// TIA Portal V19 export
FUNCTION_BLOCK "A0301_Spintore_Lat_FB"   // FB59, LAD
TITLE = == GESTIONE DELLA STAZIONE P5 ==
// stored: MemoryReserve 100, SetENOAutomatically false
   VAR_INPUT
      AreaInterface { ExternalAccessible := 'False'; ExternalVisible := 'False'; ExternalWritable := 'False'} : "AreaInterface";
      ZSI { ExternalAccessible := 'False'; ExternalVisible := 'False'; ExternalWritable := 'False'} : "udt_ZoneSafetyInterface";
      DSI { ExternalAccessible := 'False'; ExternalVisible := 'False'; ExternalWritable := 'False'} : "udt_DeviceSafetyInterface";
      DataIn : Struct
         OP_Rest_PB : Bool;
         OP_Work_PB : Bool;
         Orz_1_AnalSens : Int;
         Orz_2_AnalSens : Int;
      END_STRUCT;
      CIn { ExternalAccessible := 'False'; ExternalVisible := 'False'; ExternalWritable := 'False'} : Struct
         Manager_SpinLat_1 : "ValveMachine_Manager";
         Manager_SpinLat_2 : "ValveMachine_Manager";
         Manager_Sollevatori : "ValveMachine_Manager";
         SemiAut_Pb : Bool;
         P4 : Struct
            Fermi : "ValveMachine_COut";
         END_STRUCT;
         P5 : Struct
            SpintoreLong : Struct   // Spintore Longitudinale
               Ax_Sts : Struct
                  PosAttesa_Reached : Bool;
                  PosFineSpinta_Reached : Bool;
               END_STRUCT;
               Spintore : "ValveMachine_COut";
               Ax : "Positioning_EPOS_Machine_COut";
               Vrt : "ValveMachine_COut";
               Orz : "ValveMachine_COut";
            END_STRUCT;
         END_STRUCT;
         Trasporto : "SpeedMachine_COut";
      END_STRUCT;
      Config : Struct
         Vrt_1 : "ValveMachine_Config";
         Orz_1 : "ValveMachine_Config";
         Vrt_2 : "ValveMachine_Config";
         Orz_2 : "ValveMachine_Config";
         Sollevatori : Array[1..7] of "ValveMachine_Config";
         QuotaIngombro_SpinLat2 : Real := 2700.0;
         QuotaIngombro_SpinLat1 { ExternalWritable := 'False'} : Real := 770.0;
         DelayMissingCondition : Time;
      END_STRUCT;
   END_VAR
   VAR_OUTPUT
      MachineInterface : "MachineInterface";
      COut : Struct
         Spin_Lat1 : Struct
            Standstill : Bool;
            Rest_CheckNext : Bool;
            Work_CheckNext : Bool;
            Rest : Bool;
            Work : Bool;
         END_STRUCT;
         Spin_Lat2 : Struct
            Standstill : Bool;
            Rest_CheckNext : Bool;
            Work_CheckNext : Bool;
            Rest : Bool;
            Work : Bool;
         END_STRUCT;
         Vrt_1 : "ValveMachine_COut";
         Orz_1 : "ValveMachine_COut";
         Vrt_2 : "ValveMachine_COut";
         Orz_2 : "ValveMachine_COut";
         Sollevatori : "ValveMachine_COut";
      END_STRUCT;
   END_VAR
   VAR_IN_OUT
      Spin_Lat_1 : Struct
         Par : "Analogic_SensorManagement_Par";
         Data : Struct
            Sens : "Analogic_SensorManagement_Data";
            HMI : "HMI_Preset";
         END_STRUCT;
         Par_Mach : "A0301_Mach_Sens_Par";
      END_STRUCT;
      Spin_Lat_2 : Struct
         Par : "Analogic_SensorManagement_Par";
         Data : Struct
            Sens : "Analogic_SensorManagement_Data";
            HMI : "HMI_Preset";
         END_STRUCT;
         Par_Mach : "A0301_Mach_Sens_Par";
      END_STRUCT;
   END_VAR
   VAR
      Alarm : Struct
         Vrt_1 : "ValveAlr";
         Orz_1 { S7_SetPoint := 'True'} : "ValveAlr";
         Orz_1_AnalSens_Issue : Bool;
         Vrt_2 : "ValveAlr";
         Orz_2 { S7_SetPoint := 'True'} : "ValveAlr";
         Orz_2_AnalSens_Issue : Bool;
         Sollevatori : Array[1..7] of "ValveAlr";
         Finestre : Struct
            SpinLat2_SpinLong_Stop : Bool;   // Allarme Spintore longitudinale a ridosso dello Spintore laterale 2 che non si è abbassato
            SpinLat1_SpinLong_Stop : Bool;   // Allarme Spintore longitudinale a ridosso dello Spintore laterale 1 che non si è abbassato
         END_STRUCT;
      END_STRUCT;
      Warning : Struct
         Vrt_1 : "ValveMachine_Wng";
         Orz_1 { S7_SetPoint := 'True'} : "ValveMachine_Wng";
         Orz_1_AnalSens { ExternalAccessible := 'False'; ExternalVisible := 'False'; ExternalWritable := 'False'} : "Analogic_SensorManagement_Warning";
         Vrt_2 : "ValveMachine_Wng";
         Orz_2 { S7_SetPoint := 'True'} : "ValveMachine_Wng";
         Orz_2_AnalSens { ExternalAccessible := 'False'; ExternalVisible := 'False'; ExternalWritable := 'False'} : "Analogic_SensorManagement_Warning";
         Sollevatori : Array[1..7] of "ValveMachine_Wng";
         Finestre : Struct
            SpinLat2_SpinLong_Stop : Bool;   // Allarme Spintore longitudinale a ridosso dello Spintore laterale 2 che non si è abbassato
            SpinLat1_SpinLong_Stop : Bool;   // Allarme Spintore longitudinale a ridosso dello Spintore laterale 1 che non si è abbassato
         END_STRUCT;
         OP_REST_MissingCnd : Bool;   // Mancanza comando arresto
         OP_WORK_MissingCnd : Bool;   // Mancanza consenso lavoro
      END_STRUCT;
      HMI : Struct
         Selection : Array[1..6] of Bool;   // 0=Disable / 1=Enable Pin
         Sollevatori_Sts { S7_SetPoint := 'True'} : "UDT_HMI-Sts_ValvePosA0301";
         "SpinLat1&2_Sts" { S7_SetPoint := 'True'} : "UDT_HMI-Sts_ValvePosA0301";
         "SpinLat1&2_Vrt_Sts" { S7_SetPoint := 'True'} : "UDT_HMI-Sts_ValvePosA0301";
         "SpinLat1&2_Orz_Sts" { S7_SetPoint := 'True'} : "UDT_HMI-Sts_ValvePosA0301";
         Orz_AnalSens_PB_Preset { ExternalAccessible := 'False'; ExternalVisible := 'False'; ExternalWritable := 'False'} : Bool;   // Pulsante Preset value
         Orz_AnalSens_Preset_Value : LReal;
      END_STRUCT;
      Sts : Struct
         "SpinLat1&2_Alarm" : Bool;
         "SpinLat1&2_Vrt_AlarmPresence" : Bool;
         "SpinLat1&2_Orz_AlarmPresence" : Bool;
         Sollevatori_AlarmPresence : Bool;
         OP_CanMoveFreely : Bool;
         OP_Rest_Cnd : Bool;
         Op_Work_Cnd : Bool;
         Beam : Struct
            H_B : Real;
            Len_Meas : Real;
            P_U_PLen : Real;
            P_L_PLen : Real;
         END_STRUCT;
         "En/Dis_SpinLat_2" : Bool;   // 1=Enable / 0=Disable
      END_STRUCT;
      Ctrl : Struct
         OP_Rest_Man : Bool;
         OP_Work_Man : Bool;
         OP_Rest_Aut : Bool;
         OP_Work_Aut : Bool;
         OP_Rest : Bool;
         OP_Work : Bool;
      END_STRUCT;
      Vrt_1 : "ValveMachine_FB";
      Orz_1 { S7_SetPoint := 'True'} : "ValveMachine_FB";
      Orz_1_AnalSens { S7_SetPoint := 'True'} : "Analogic_SensorManagement";
      Vrt_2 : "ValveMachine_FB";
      Orz_2 { S7_SetPoint := 'True'} : "ValveMachine_FB";
      Orz_2_AnalSens { S7_SetPoint := 'True'} : "Analogic_SensorManagement";
      Sollevatori : Array[1..6] of "ValveMachine_FB";
      AUX : Struct
         OP_Rest_PB : Bool;
         OP_Work_PB : Bool;
      END_STRUCT;
      TON_OP_REST_MissingCnd { S7_SetPoint := 'True'} : TON_TIME;
      TON_OP_WORK_MissingCnd { S7_SetPoint := 'True'} : TON_TIME;
      Finestre : Struct
         Quota_SpinLat2_Rest : Real;   // Quota per comando riposo SpintoreLaterale 2
         Quota_SpinLat1_Rest : Real;   // Quota per comando riposo SpintoreLaterale 1
         RestCnd_Vrt_1 : Bool;   // Spintore longitudinale a ridosso dello Spintore laterale 1 - Comando riposo
         RestCnd_Vrt_2 : Bool;   // Spintore longitudinale a ridosso dello Spintore laterale 2 - Comando riposo
      END_STRUCT;
   END_VAR
   VAR_TEMP
      PE : Struct
         OP_Rest_PB : Bool;
         OP_Work_PB : Bool;
      END_STRUCT;
   END_VAR
   VAR CONSTANT
      Offset_SpinLat2_Rest : Real := 50.0;   // Offset calcolato da quota ingombro Spintore Laterale2 per abbassarlo
      Offset_SpinLat1_Rest : Real := 50.0;   // Offset calcolato da quota ingombro Spintore Laterale1 per abbassarlo
   END_VAR
   VAR_TEMP   // added for the SCL form of the ladder/FBD networks
      _w1 : Bool;
      _w2 : Bool;
      _w3 : Bool;
      _w4 : Bool;
      _w5 : Bool;
      _w6 : Bool;
      _w7 : Bool;
      _w8 : Bool;
   END_VAR
BEGIN

REGION Network 1 (SCL): Reset allarmi
   IF #AreaInterface.RstAlarms THEN
       #Alarm.Orz_1_AnalSens_Issue := FALSE;
       #Alarm.Orz_2_AnalSens_Issue := FALSE;
   END_IF;

   IF #AreaInterface.RstAlarms AND #Vrt_2.COut.Rest AND #Orz_2.COut.Rest THEN
       #Alarm.Finestre.SpinLat2_SpinLong_Stop := 0;
       #Warning.Finestre.SpinLat2_SpinLong_Stop := 0;
   END_IF;

   IF #AreaInterface.RstAlarms AND #Vrt_1.COut.Rest AND #Orz_1.COut.Rest THEN
       #Alarm.Finestre.SpinLat1_SpinLong_Stop := 0;
       #Warning.Finestre.SpinLat1_SpinLong_Stop := 0;
   END_IF;
END_REGION

REGION Network 2: <+>
END_REGION

REGION Network 3: CONTROLLO -
END_REGION

REGION Network 4 (SCL): CONTROLLO - Finestre di ingombro & Controlli di posizione

   // Finestra ingombro SPINTORE LATERALE 2
   #Finestre.Quota_SpinLat2_Rest := #Config.QuotaIngombro_SpinLat2 - #Offset_SpinLat2_Rest;

   // Se ho lo Spintore longitudinale in movimento ed entro dentro la finestra abbasso lo Spintore laterale 2 prima di arrivarci addosso
   // //
   IF #Sts.Beam.Len_Meas <= 2700.0 THEN
       #Sts."En/Dis_SpinLat_2" := FALSE;

   ELSE
       #Sts."En/Dis_SpinLat_2" := TRUE;
       #Warning.Finestre.SpinLat2_SpinLong_Stop := FALSE;
   END_IF;

   //Se arrivo in quota ingombro spintore lat. 2 mando a riposo attivando il cmd finestra
   IF  #Finestre.Quota_SpinLat2_Rest <= #CIn.P5.SpintoreLong.Ax.ActualPosition THEN
       #Finestre.RestCnd_Vrt_2 := TRUE;
   ELSE
       #Finestre.RestCnd_Vrt_2 := FALSE;
   END_IF;

   // Se supero la quota di riposo Spintore Laterale 2 e non sono ancora a riposo con Spintore Laterale attivo warning
   IF #Finestre.Quota_SpinLat2_Rest < #CIn.P5.SpintoreLong.Ax.ActualPosition AND NOT #Vrt_2.COut.Rest THEN
       #Warning.Finestre.SpinLat2_SpinLong_Stop := TRUE;
   END_IF;

   //Se vado a riposo con spin. lat 2 resetto warning 
   IF (#Vrt_2.COut.Rest AND #Orz_2.COut.Rest) THEN
       #Warning.Finestre.SpinLat2_SpinLong_Stop := FALSE;
   END_IF;

   // Finestra ingombro SPINTORE LATERALE 1
   #Finestre.Quota_SpinLat1_Rest := #Config.QuotaIngombro_SpinLat1 - #Offset_SpinLat1_Rest;

   // Se ho lo Spintore longitudinale in movimento ed entro dentro la finestra abbasso lo Spintore laterale 1 prima di arrivarci addosso

   //Se arrivo in quota ingombro spintore lat. 1 mando a riposo attivando il cmd finestra 
   IF #Finestre.Quota_SpinLat1_Rest <= #CIn.P5.SpintoreLong.Ax.ActualPosition  THEN
       #Finestre.RestCnd_Vrt_1 := TRUE;
   ELSE
       #Finestre.RestCnd_Vrt_1 := FALSE;
   END_IF;

   // Se supero la quota di riposo Spintore Laterale 1 e non sono ancora a riposo con Spintore Laterale attivo warning
   IF #Finestre.Quota_SpinLat1_Rest < #CIn.P5.SpintoreLong.Ax.ActualPosition AND NOT #Vrt_1.COut.Rest THEN
       #Warning.Finestre.SpinLat1_SpinLong_Stop := TRUE;
   END_IF;

   //Se vado a riposo con spin. lat 2 resetto warning 
   IF (#Vrt_1.COut.Rest AND #Orz_1.COut.Rest) THEN
       #Warning.Finestre.SpinLat2_SpinLong_Stop := FALSE;

   END_IF;
END_REGION

REGION Network 5: <+>
END_REGION

REGION Network 6: Operazione può muoversi liberamente perchè non sposta nessun BEAM
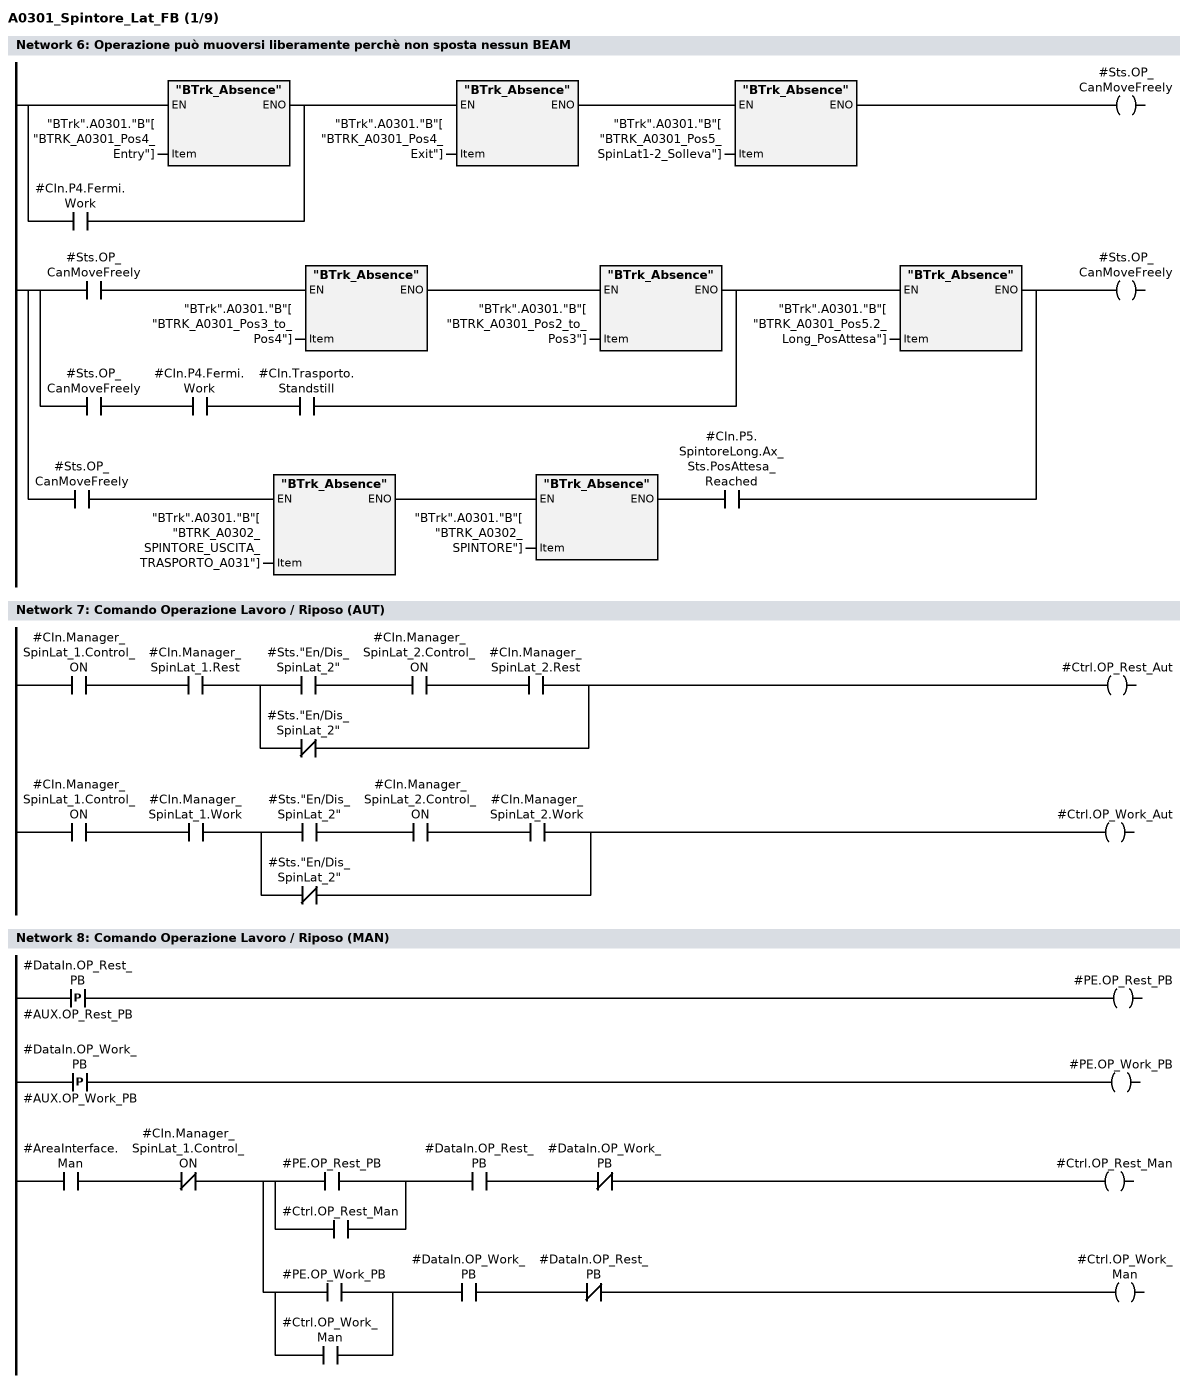
   RUNG wire#powerrail
      "BTrk_Absence"(Item := "BTrk".A0301."B"["BTRK_A0301_Pos4_Entry"])
      wire#w1
      "BTrk_Absence"(Item := "BTrk".A0301."B"["BTRK_A0301_Pos4_Exit"])
      "BTrk_Absence"(Item := "BTrk".A0301."B"["BTRK_A0301_Pos5_SpinLat1-2_Solleva"])
      Coil( #Sts.OP_CanMoveFreely )
   END_RUNG
   RUNG wire#powerrail
      Contact( #CIn.P4.Fermi.Work )
   END_RUNG wire#w1
   RUNG wire#powerrail
      Contact( #Sts.OP_CanMoveFreely )
      "BTrk_Absence"(Item := "BTrk".A0301."B"["BTRK_A0301_Pos3_to_Pos4"])
      "BTrk_Absence"(Item := "BTrk".A0301."B"["BTRK_A0301_Pos2_to_Pos3"])
      wire#w2
      "BTrk_Absence"(Item := "BTrk".A0301."B"["BTRK_A0301_Pos5.2_Long_PosAttesa"])
      wire#w3
      Coil( #Sts.OP_CanMoveFreely )
   END_RUNG
   RUNG wire#powerrail
      Contact( #Sts.OP_CanMoveFreely )
      Contact( #CIn.P4.Fermi.Work )
      Contact( #CIn.Trasporto.Standstill )
   END_RUNG wire#w2
   RUNG wire#powerrail
      Contact( #Sts.OP_CanMoveFreely )
      "BTrk_Absence"(Item := "BTrk".A0301."B"["BTRK_A0302_SPINTORE_USCITA_TRASPORTO_A031"])
      "BTrk_Absence"(Item := "BTrk".A0301."B"["BTRK_A0302_SPINTORE"])
      Contact( #CIn.P5.SpintoreLong.Ax_Sts.PosAttesa_Reached )
   END_RUNG wire#w3
   // the same network as SCL:
   "BTrk_Absence"(Item := "BTrk".A0301."B"["BTRK_A0301_Pos4_Entry"], ENO => #_w1);
   "BTrk_Absence"(EN := #_w1 OR #CIn.P4.Fermi.Work,
                  Item := "BTrk".A0301."B"["BTRK_A0301_Pos4_Exit"],
                  ENO => #_w2);
   "BTrk_Absence"(EN := #_w2, Item := "BTrk".A0301."B"["BTRK_A0301_Pos5_SpinLat1-2_Solleva"], ENO => #_w3);
   #Sts.OP_CanMoveFreely := #_w3;
   "BTrk_Absence"(EN := #Sts.OP_CanMoveFreely, Item := "BTrk".A0301."B"["BTRK_A0301_Pos3_to_Pos4"], ENO => #_w4);
   "BTrk_Absence"(EN := #_w4, Item := "BTrk".A0301."B"["BTRK_A0301_Pos2_to_Pos3"], ENO => #_w5);
   "BTrk_Absence"(EN := #_w5 OR (#Sts.OP_CanMoveFreely AND #CIn.P4.Fermi.Work AND #CIn.Trasporto.Standstill),
                  Item := "BTrk".A0301."B"["BTRK_A0301_Pos5.2_Long_PosAttesa"],
                  ENO => #_w6);
   "BTrk_Absence"(EN := #Sts.OP_CanMoveFreely,
                  Item := "BTrk".A0301."B"["BTRK_A0302_SPINTORE_USCITA_TRASPORTO_A031"],
                  ENO => #_w7);
   "BTrk_Absence"(EN := #_w7, Item := "BTrk".A0301."B"["BTRK_A0302_SPINTORE"], ENO => #_w8);
   #Sts.OP_CanMoveFreely := #_w6 OR (#_w8 AND #CIn.P5.SpintoreLong.Ax_Sts.PosAttesa_Reached);
END_REGION

REGION Network 7: Comando Operazione Lavoro / Riposo (AUT)
   RUNG wire#powerrail
      Contact( #CIn.Manager_SpinLat_1.Control_ON )
      Contact( #CIn.Manager_SpinLat_1.Rest )
      wire#w1
      Contact( #Sts."En/Dis_SpinLat_2" )
      Contact( #CIn.Manager_SpinLat_2.Control_ON )
      Contact( #CIn.Manager_SpinLat_2.Rest )
      wire#w2
      Coil( #Ctrl.OP_Rest_Aut )
   END_RUNG
   RUNG wire#w1
      I_Contact( #Sts."En/Dis_SpinLat_2" )
   END_RUNG wire#w2
   RUNG wire#powerrail
      Contact( #CIn.Manager_SpinLat_1.Control_ON )
      Contact( #CIn.Manager_SpinLat_1.Work )
      wire#w3
      Contact( #Sts."En/Dis_SpinLat_2" )
      Contact( #CIn.Manager_SpinLat_2.Control_ON )
      Contact( #CIn.Manager_SpinLat_2.Work )
      wire#w4
      Coil( #Ctrl.OP_Work_Aut )
   END_RUNG
   RUNG wire#w3
      I_Contact( #Sts."En/Dis_SpinLat_2" )
   END_RUNG wire#w4
   // the same network as SCL:
   #Ctrl.OP_Rest_Aut := #CIn.Manager_SpinLat_1.Control_ON AND #CIn.Manager_SpinLat_1.Rest AND ((#Sts."En/Dis_SpinLat_2" AND #CIn.Manager_SpinLat_2.Control_ON AND #CIn.Manager_SpinLat_2.Rest) OR NOT #Sts."En/Dis_SpinLat_2");
   #Ctrl.OP_Work_Aut := #CIn.Manager_SpinLat_1.Control_ON AND #CIn.Manager_SpinLat_1.Work AND ((#Sts."En/Dis_SpinLat_2" AND #CIn.Manager_SpinLat_2.Control_ON AND #CIn.Manager_SpinLat_2.Work) OR NOT #Sts."En/Dis_SpinLat_2");
END_REGION

REGION Network 8: Comando Operazione Lavoro / Riposo (MAN)
   RUNG wire#powerrail
      P_Contact(operand := #DataIn.OP_Rest_PB, bit := #AUX.OP_Rest_PB)
      Coil( #PE.OP_Rest_PB )
   END_RUNG
   RUNG wire#powerrail
      P_Contact(operand := #DataIn.OP_Work_PB, bit := #AUX.OP_Work_PB)
      Coil( #PE.OP_Work_PB )
   END_RUNG
   RUNG wire#powerrail
      Contact( #AreaInterface.Man )
      I_Contact( #CIn.Manager_SpinLat_1.Control_ON )
      wire#w1
      Contact( #PE.OP_Rest_PB )
      wire#w2
      Contact( #DataIn.OP_Rest_PB )
      I_Contact( #DataIn.OP_Work_PB )
      Coil( #Ctrl.OP_Rest_Man )
   END_RUNG
   RUNG wire#w1
      Contact( #Ctrl.OP_Rest_Man )
   END_RUNG wire#w2
   RUNG wire#w1
      Contact( #PE.OP_Work_PB )
      wire#w3
      Contact( #DataIn.OP_Work_PB )
      I_Contact( #DataIn.OP_Rest_PB )
      Coil( #Ctrl.OP_Work_Man )
   END_RUNG
   RUNG wire#w1
      Contact( #Ctrl.OP_Work_Man )
   END_RUNG wire#w3
   // the same network as SCL:
   #_w1 := #DataIn.OP_Rest_PB AND NOT #AUX.OP_Rest_PB;   // rising edge of #DataIn.OP_Rest_PB
   #AUX.OP_Rest_PB := #DataIn.OP_Rest_PB;
   #PE.OP_Rest_PB := #_w1;
   #_w2 := #DataIn.OP_Work_PB AND NOT #AUX.OP_Work_PB;   // rising edge of #DataIn.OP_Work_PB
   #AUX.OP_Work_PB := #DataIn.OP_Work_PB;
   #PE.OP_Work_PB := #_w2;
   #_w3 := #AreaInterface.Man AND NOT #CIn.Manager_SpinLat_1.Control_ON;
   #Ctrl.OP_Rest_Man := #_w3 AND (#PE.OP_Rest_PB OR #Ctrl.OP_Rest_Man) AND #DataIn.OP_Rest_PB AND NOT #DataIn.OP_Work_PB;
   #Ctrl.OP_Work_Man := #_w3 AND (#PE.OP_Work_PB OR #Ctrl.OP_Work_Man) AND #DataIn.OP_Work_PB AND NOT #DataIn.OP_Rest_PB;
END_REGION

REGION Network 9: Cumulativo Operazione Lavoro / Riposo (ALL)
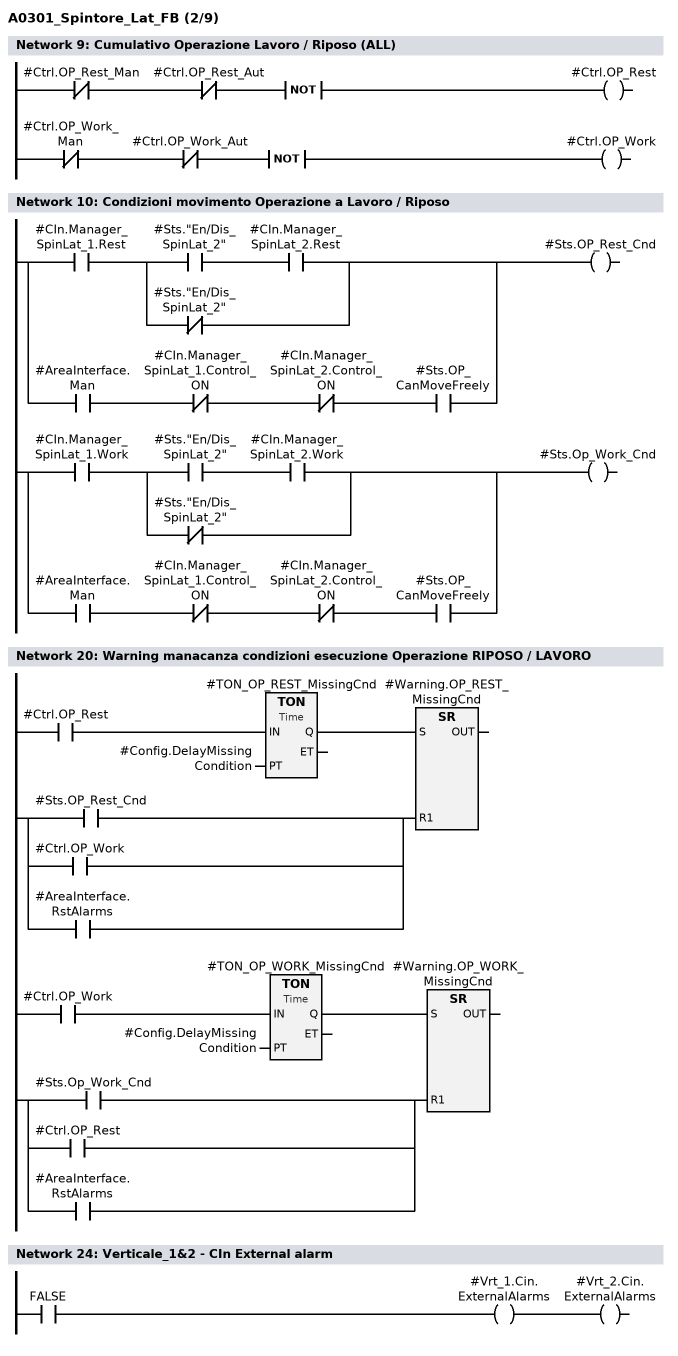
   RUNG wire#powerrail
      I_Contact( #Ctrl.OP_Rest_Man )
      I_Contact( #Ctrl.OP_Rest_Aut )
      Not()
      Coil( #Ctrl.OP_Rest )
   END_RUNG
   RUNG wire#powerrail
      I_Contact( #Ctrl.OP_Work_Man )
      I_Contact( #Ctrl.OP_Work_Aut )
      Not()
      Coil( #Ctrl.OP_Work )
   END_RUNG
   // the same network as SCL:
   #Ctrl.OP_Rest := NOT (NOT #Ctrl.OP_Rest_Man AND NOT #Ctrl.OP_Rest_Aut);
   #Ctrl.OP_Work := NOT (NOT #Ctrl.OP_Work_Man AND NOT #Ctrl.OP_Work_Aut);
END_REGION

REGION Network 10: Condizioni movimento Operazione a Lavoro / Riposo
   RUNG wire#powerrail
      Contact( #CIn.Manager_SpinLat_1.Rest )
      wire#w1
      Contact( #Sts."En/Dis_SpinLat_2" )
      Contact( #CIn.Manager_SpinLat_2.Rest )
      wire#w2
      Coil( #Sts.OP_Rest_Cnd )
   END_RUNG
   RUNG wire#w1
      I_Contact( #Sts."En/Dis_SpinLat_2" )
   END_RUNG wire#w2
   RUNG wire#powerrail
      Contact( #AreaInterface.Man )
      I_Contact( #CIn.Manager_SpinLat_1.Control_ON )
      I_Contact( #CIn.Manager_SpinLat_2.Control_ON )
      Contact( #Sts.OP_CanMoveFreely )
   END_RUNG wire#w2
   RUNG wire#powerrail
      Contact( #CIn.Manager_SpinLat_1.Work )
      wire#w3
      Contact( #Sts."En/Dis_SpinLat_2" )
      Contact( #CIn.Manager_SpinLat_2.Work )
      wire#w4
      Coil( #Sts.Op_Work_Cnd )
   END_RUNG
   RUNG wire#w3
      I_Contact( #Sts."En/Dis_SpinLat_2" )
   END_RUNG wire#w4
   RUNG wire#powerrail
      Contact( #AreaInterface.Man )
      I_Contact( #CIn.Manager_SpinLat_1.Control_ON )
      I_Contact( #CIn.Manager_SpinLat_2.Control_ON )
      Contact( #Sts.OP_CanMoveFreely )
   END_RUNG wire#w4
   // the same network as SCL:
   #Sts.OP_Rest_Cnd := (#CIn.Manager_SpinLat_1.Rest AND ((#Sts."En/Dis_SpinLat_2" AND #CIn.Manager_SpinLat_2.Rest) OR NOT #Sts."En/Dis_SpinLat_2")) OR (#AreaInterface.Man AND NOT #CIn.Manager_SpinLat_1.Control_ON AND NOT #CIn.Manager_SpinLat_2.Control_ON AND #Sts.OP_CanMoveFreely);
   #Sts.Op_Work_Cnd := (#CIn.Manager_SpinLat_1.Work AND ((#Sts."En/Dis_SpinLat_2" AND #CIn.Manager_SpinLat_2.Work) OR NOT #Sts."En/Dis_SpinLat_2")) OR (#AreaInterface.Man AND NOT #CIn.Manager_SpinLat_1.Control_ON AND NOT #CIn.Manager_SpinLat_2.Control_ON AND #Sts.OP_CanMoveFreely);
END_REGION

REGION Network 11: <+>
END_REGION

REGION Network 12 (SCL): Verticale + Orizzontale 1 - Cin Manager (Esecuzione sequenza comandi)
   #Vrt_1.Cin.Manager.Control_ON := #Orz_1.Cin.Manager.Control_ON := #CIn.Manager_SpinLat_1.Control_ON;

   #Vrt_1.Cin.Manager.Rest := FALSE;
   #Vrt_1.Cin.Manager.Work := FALSE;
   #Orz_1.Cin.Manager.Rest := FALSE;
   #Orz_1.Cin.Manager.Work := FALSE;


       IF (#Ctrl.OP_Rest AND #Sts.OP_Rest_Cnd) OR #Finestre.RestCnd_Vrt_1 THEN

           #Orz_1.Cin.Manager.Rest := #Vrt_1.Cin.Manager.Rest := TRUE;

       ELSIF (#Ctrl.OP_Work AND #Sts.Op_Work_Cnd) AND NOT #Finestre.RestCnd_Vrt_1 THEN

           #Orz_1.Cin.Manager.Work := #Vrt_1.Cin.Manager.Work := TRUE;

       END_IF;
END_REGION

REGION Network 13 (SCL): Verticale + Orizzontale1 - CIn Abilitazioni Stop Manager
   #Vrt_1.Cin.Manager.EnableStopDoorOpeningReq := #Orz_1.Cin.Manager.EnableStopDoorOpeningReq := #CIn.Manager_SpinLat_1.EnableStopDoorOpeningReq;

   #Vrt_1.Cin.Manager.EnableStopInPhase := #Orz_1.Cin.Manager.EnableStopInPhase := #CIn.Manager_SpinLat_1.EnableStopInPhase;

   #Vrt_1.Cin.Manager.EnableStopProgrammed := #Orz_1.Cin.Manager.EnableStopProgrammed := #CIn.Manager_SpinLat_1.EnableStopProgrammed;
END_REGION

REGION Network 14 (SCL): Verticale + Orizzontale 2 - Cin Manager (Esecuzione sequenza comandi)
   // Controllo della misura in lunghezza del Beam per sapere se abilitare il secondo spintore
   //
   #Vrt_2.Cin.Manager.Control_ON := #Orz_2.Cin.Manager.Control_ON := #CIn.Manager_SpinLat_2.Control_ON;
   //
   #Vrt_2.Cin.Manager.Rest := FALSE;
   #Vrt_2.Cin.Manager.Work := FALSE;
   #Orz_2.Cin.Manager.Rest := FALSE;
   #Orz_2.Cin.Manager.Work := FALSE;



   IF (#Ctrl.OP_Rest AND #Sts.OP_Rest_Cnd )OR #Finestre.RestCnd_Vrt_2 OR #Warning.Finestre.SpinLat2_SpinLong_Stop THEN

           #Orz_2.Cin.Manager.Rest := #Vrt_2.Cin.Manager.Rest := TRUE;

       ELSIF (#Ctrl.OP_Work AND #Sts.Op_Work_Cnd) AND #Sts."En/Dis_SpinLat_2" AND NOT #Finestre.RestCnd_Vrt_2  THEN

           #Orz_2.Cin.Manager.Work := #Vrt_2.Cin.Manager.Work := TRUE;

       END_IF;
END_REGION

REGION Network 15 (SCL): Verticale + Orizzontale 2 - CIn Abilitazioni Stop Manager
   #Vrt_2.Cin.Manager.EnableStopDoorOpeningReq := #Orz_2.Cin.Manager.EnableStopDoorOpeningReq := #CIn.Manager_SpinLat_2.EnableStopDoorOpeningReq;

   #Vrt_2.Cin.Manager.EnableStopInPhase := #Orz_2.Cin.Manager.EnableStopInPhase := #CIn.Manager_SpinLat_2.EnableStopInPhase;

   #Vrt_2.Cin.Manager.EnableStopProgrammed := #Orz_2.Cin.Manager.EnableStopProgrammed := #CIn.Manager_SpinLat_2.EnableStopProgrammed;
END_REGION

REGION Network 16: <+>
END_REGION

REGION Network 17 (SCL): S[1...7] Sollevatori - Cin Manager Comando arresto / lavoro
   //
   #Sollevatori[1].Cin.Manager.Rest := FALSE;
   #Sollevatori[2].Cin.Manager.Rest := FALSE;
   #Sollevatori[3].Cin.Manager.Rest := FALSE;
   #Sollevatori[4].Cin.Manager.Rest := FALSE;
   #Sollevatori[5].Cin.Manager.Rest := FALSE;
   #Sollevatori[6].Cin.Manager.Rest := FALSE;
   //************************************
   #Sollevatori[1].Cin.Manager.Work := FALSE;
   #Sollevatori[2].Cin.Manager.Work := FALSE;
   #Sollevatori[3].Cin.Manager.Work := FALSE;
   #Sollevatori[4].Cin.Manager.Work := FALSE;
   #Sollevatori[5].Cin.Manager.Work := FALSE;
   #Sollevatori[6].Cin.Manager.Work := FALSE;
   //
   // CIn Manager  Control ON se ho un richiesta di comando attiva
   IF #AreaInterface.Aut OR #CIn.SemiAut_Pb THEN
       #Sollevatori[1].Cin.Manager.Control_ON := TRUE;
       #Sollevatori[2].Cin.Manager.Control_ON := TRUE;
       #Sollevatori[3].Cin.Manager.Control_ON := TRUE;
       #Sollevatori[4].Cin.Manager.Control_ON := TRUE;
       #Sollevatori[5].Cin.Manager.Control_ON := TRUE;
       #Sollevatori[6].Cin.Manager.Control_ON := TRUE;
   ELSE
       #Sollevatori[1].Cin.Manager.Control_ON := FALSE;
       #Sollevatori[2].Cin.Manager.Control_ON := FALSE;
       #Sollevatori[3].Cin.Manager.Control_ON := FALSE;
       #Sollevatori[4].Cin.Manager.Control_ON := FALSE;
       #Sollevatori[5].Cin.Manager.Control_ON := FALSE;
       #Sollevatori[6].Cin.Manager.Control_ON := FALSE;
   END_IF;

   // CIn Manager Rest se ho un richiesta di comando arresto attiva
   IF #CIn.Manager_Sollevatori.Rest THEN

       #Sollevatori[1].Cin.Manager.Rest := TRUE;
       #Sollevatori[2].Cin.Manager.Rest := TRUE;
       #Sollevatori[3].Cin.Manager.Rest := TRUE;
       #Sollevatori[4].Cin.Manager.Rest := TRUE;
       #Sollevatori[5].Cin.Manager.Rest := TRUE;
       #Sollevatori[6].Cin.Manager.Rest := TRUE;

       // CIn Manager Work se ho un richiesta di comando lavoro attiva   
       ELSIF #CIn.Manager_Sollevatori.Work THEN

       #Sollevatori[1].Cin.Manager.Work := TRUE;
       #Sollevatori[2].Cin.Manager.Work := TRUE;
       #Sollevatori[3].Cin.Manager.Work := TRUE;
       #Sollevatori[4].Cin.Manager.Work := TRUE;
       #Sollevatori[5].Cin.Manager.Work := TRUE;
       #Sollevatori[6].Cin.Manager.Work := TRUE;

   END_IF;
END_REGION

REGION Network 18 (SCL): S[1...7] Sollevatori - CIn Abilitazioni Stop Manager
   //
   // CIn Manager Stop per richiesta apertura safety
   IF #CIn.Manager_SpinLat_1.EnableStopDoorOpeningReq THEN
       #Sollevatori[1].Cin.Manager.EnableStopDoorOpeningReq := TRUE;
       #Sollevatori[2].Cin.Manager.EnableStopDoorOpeningReq := TRUE;
       #Sollevatori[3].Cin.Manager.EnableStopDoorOpeningReq := TRUE;
       #Sollevatori[4].Cin.Manager.EnableStopDoorOpeningReq := TRUE;
       #Sollevatori[5].Cin.Manager.EnableStopDoorOpeningReq := TRUE;
       #Sollevatori[6].Cin.Manager.EnableStopDoorOpeningReq := TRUE;

   ELSE
       #Sollevatori[1].Cin.Manager.EnableStopDoorOpeningReq := FALSE;
       #Sollevatori[2].Cin.Manager.EnableStopDoorOpeningReq := FALSE;
       #Sollevatori[3].Cin.Manager.EnableStopDoorOpeningReq := FALSE;
       #Sollevatori[4].Cin.Manager.EnableStopDoorOpeningReq := FALSE;
       #Sollevatori[5].Cin.Manager.EnableStopDoorOpeningReq := FALSE;
       #Sollevatori[6].Cin.Manager.EnableStopDoorOpeningReq := FALSE;

   END_IF;
   // CIn Manager Stop in fase delle macchine precedenti
   IF #CIn.Manager_SpinLat_1.EnableStopInPhase THEN
       #Sollevatori[1].Cin.Manager.EnableStopInPhase := TRUE;
       #Sollevatori[2].Cin.Manager.EnableStopInPhase := TRUE;
       #Sollevatori[3].Cin.Manager.EnableStopInPhase := TRUE;
       #Sollevatori[4].Cin.Manager.EnableStopInPhase := TRUE;
       #Sollevatori[5].Cin.Manager.EnableStopInPhase := TRUE;
       #Sollevatori[6].Cin.Manager.EnableStopInPhase := TRUE;

   ELSE
       #Sollevatori[1].Cin.Manager.EnableStopInPhase := FALSE;
       #Sollevatori[2].Cin.Manager.EnableStopInPhase := FALSE;
       #Sollevatori[3].Cin.Manager.EnableStopInPhase := FALSE;
       #Sollevatori[4].Cin.Manager.EnableStopInPhase := FALSE;
       #Sollevatori[5].Cin.Manager.EnableStopInPhase := FALSE;
       #Sollevatori[6].Cin.Manager.EnableStopInPhase := FALSE;

   END_IF;

   // CIn Manager Stop programmato configurabile a piacere
   IF #CIn.Manager_SpinLat_1.EnableStopProgrammed THEN
       #Sollevatori[1].Cin.Manager.EnableStopProgrammed := TRUE;
       #Sollevatori[2].Cin.Manager.EnableStopProgrammed := TRUE;
       #Sollevatori[3].Cin.Manager.EnableStopProgrammed := TRUE;
       #Sollevatori[4].Cin.Manager.EnableStopProgrammed := TRUE;
       #Sollevatori[5].Cin.Manager.EnableStopProgrammed := TRUE;
       #Sollevatori[6].Cin.Manager.EnableStopProgrammed := TRUE;

   ELSE
       #Sollevatori[1].Cin.Manager.EnableStopProgrammed := FALSE;
       #Sollevatori[2].Cin.Manager.EnableStopProgrammed := FALSE;
       #Sollevatori[3].Cin.Manager.EnableStopProgrammed := FALSE;
       #Sollevatori[4].Cin.Manager.EnableStopProgrammed := FALSE;
       #Sollevatori[5].Cin.Manager.EnableStopProgrammed := FALSE;
       #Sollevatori[6].Cin.Manager.EnableStopProgrammed := FALSE;

   END_IF;
END_REGION

REGION Network 19: <+>
END_REGION

REGION Network 20: Warning manacanza condizioni esecuzione Operazione RIPOSO / LAVORO
   RUNG wire#powerrail
      Contact( #Ctrl.OP_Rest )
      { S7_Templates := "time_type := Time" } #TON_OP_REST_MissingCnd.TON(pt := #Config.DelayMissingCondition, et =>)
      S_SR(operand := #Warning.OP_REST_MissingCnd, r1 := wire#w1)
   END_RUNG
   RUNG wire#powerrail
      Contact( #Sts.OP_Rest_Cnd )
   END_RUNG wire#w1
   RUNG wire#powerrail
      Contact( #Ctrl.OP_Work )
   END_RUNG wire#w1
   RUNG wire#powerrail
      Contact( #AreaInterface.RstAlarms )
   END_RUNG wire#w1
   RUNG wire#powerrail
      Contact( #Ctrl.OP_Work )
      { S7_Templates := "time_type := Time" } #TON_OP_WORK_MissingCnd.TON(pt := #Config.DelayMissingCondition, et =>)
      S_SR(operand := #Warning.OP_WORK_MissingCnd, r1 := wire#w2)
   END_RUNG
   RUNG wire#powerrail
      Contact( #Sts.Op_Work_Cnd )
   END_RUNG wire#w2
   RUNG wire#powerrail
      Contact( #Ctrl.OP_Rest )
   END_RUNG wire#w2
   RUNG wire#powerrail
      Contact( #AreaInterface.RstAlarms )
   END_RUNG wire#w2
   // the same network as SCL:
   #TON_OP_REST_MissingCnd(IN := #Ctrl.OP_Rest, PT := #Config.DelayMissingCondition);   // TON
   IF #TON_OP_REST_MissingCnd.Q THEN
       #Warning.OP_REST_MissingCnd := TRUE;   // SR flip-flop
   END_IF;
   IF #Sts.OP_Rest_Cnd OR #Ctrl.OP_Work OR #AreaInterface.RstAlarms THEN
       #Warning.OP_REST_MissingCnd := FALSE;
   END_IF;
   #TON_OP_WORK_MissingCnd(IN := #Ctrl.OP_Work, PT := #Config.DelayMissingCondition);   // TON
   IF #TON_OP_WORK_MissingCnd.Q THEN
       #Warning.OP_WORK_MissingCnd := TRUE;   // SR flip-flop
   END_IF;
   IF #Sts.Op_Work_Cnd OR #Ctrl.OP_Rest OR #AreaInterface.RstAlarms THEN
       #Warning.OP_WORK_MissingCnd := FALSE;
   END_IF;
END_REGION

REGION Network 21: <+>
END_REGION

REGION Network 22: << GESTIONE VERTICALE >>
END_REGION

REGION Network 23 (SCL): Verticale1&2 - Data In
   // DataIn Scritti sulla CALL dell'FB
END_REGION

REGION Network 24: Verticale_1&2 - CIn External alarm
   RUNG wire#powerrail
      Contact( FALSE )
      Coil( #Vrt_1.Cin.ExternalAlarms )
      Coil( #Vrt_2.Cin.ExternalAlarms )
   END_RUNG
   // the same network as SCL:
   #Vrt_1.Cin.ExternalAlarms := FALSE;
   #Vrt_2.Cin.ExternalAlarms := FALSE;
END_REGION

REGION Network 25: Verticale_1 - Cin Ext Enable
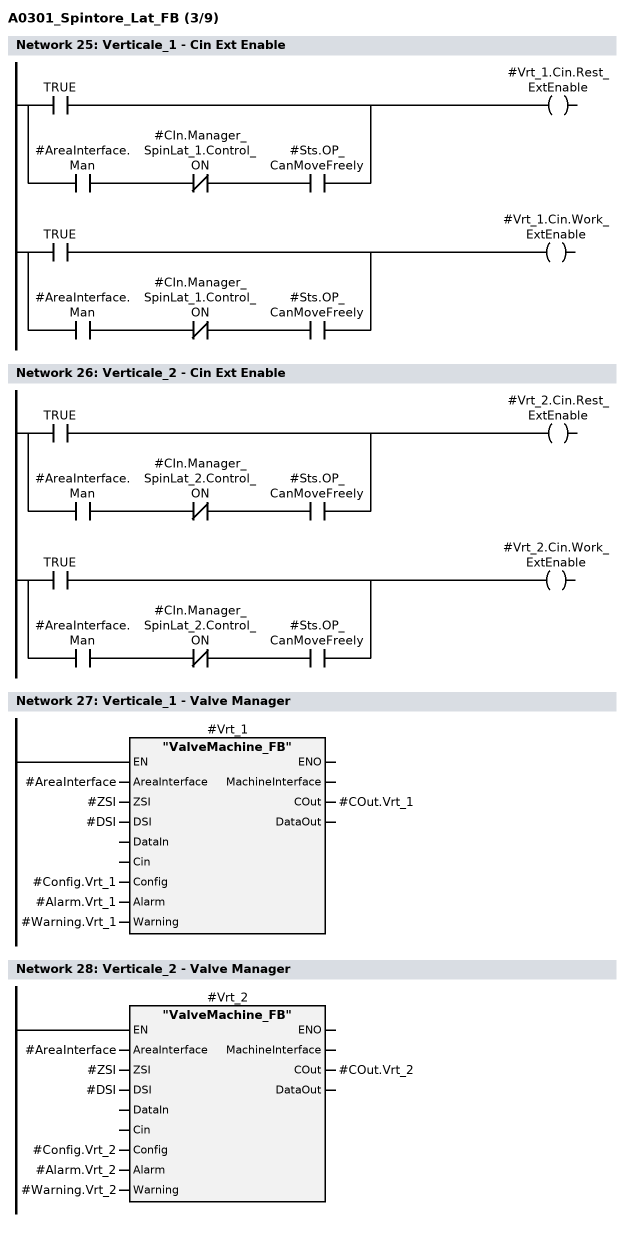
   RUNG wire#powerrail
      Contact( TRUE )
      wire#w1
      Coil( #Vrt_1.Cin.Rest_ExtEnable )
   END_RUNG
   RUNG wire#powerrail
      Contact( #AreaInterface.Man )
      I_Contact( #CIn.Manager_SpinLat_1.Control_ON )
      Contact( #Sts.OP_CanMoveFreely )
   END_RUNG wire#w1
   RUNG wire#powerrail
      Contact( TRUE )
      wire#w2
      Coil( #Vrt_1.Cin.Work_ExtEnable )
   END_RUNG
   RUNG wire#powerrail
      Contact( #AreaInterface.Man )
      I_Contact( #CIn.Manager_SpinLat_1.Control_ON )
      Contact( #Sts.OP_CanMoveFreely )
   END_RUNG wire#w2
   // the same network as SCL:
   #Vrt_1.Cin.Rest_ExtEnable := TRUE OR (#AreaInterface.Man AND NOT #CIn.Manager_SpinLat_1.Control_ON AND #Sts.OP_CanMoveFreely);
   #Vrt_1.Cin.Work_ExtEnable := TRUE OR (#AreaInterface.Man AND NOT #CIn.Manager_SpinLat_1.Control_ON AND #Sts.OP_CanMoveFreely);
END_REGION

REGION Network 26: Verticale_2 - Cin Ext Enable
   RUNG wire#powerrail
      Contact( TRUE )
      wire#w1
      Coil( #Vrt_2.Cin.Rest_ExtEnable )
   END_RUNG
   RUNG wire#powerrail
      Contact( #AreaInterface.Man )
      I_Contact( #CIn.Manager_SpinLat_2.Control_ON )
      Contact( #Sts.OP_CanMoveFreely )
   END_RUNG wire#w1
   RUNG wire#powerrail
      Contact( TRUE )
      wire#w2
      Coil( #Vrt_2.Cin.Work_ExtEnable )
   END_RUNG
   RUNG wire#powerrail
      Contact( #AreaInterface.Man )
      I_Contact( #CIn.Manager_SpinLat_2.Control_ON )
      Contact( #Sts.OP_CanMoveFreely )
   END_RUNG wire#w2
   // the same network as SCL:
   #Vrt_2.Cin.Rest_ExtEnable := TRUE OR (#AreaInterface.Man AND NOT #CIn.Manager_SpinLat_2.Control_ON AND #Sts.OP_CanMoveFreely);
   #Vrt_2.Cin.Work_ExtEnable := TRUE OR (#AreaInterface.Man AND NOT #CIn.Manager_SpinLat_2.Control_ON AND #Sts.OP_CanMoveFreely);
END_REGION

REGION Network 27: Verticale_1 - Valve Manager
   RUNG wire#powerrail
      #Vrt_1(AreaInterface := #AreaInterface, ZSI := #ZSI, DSI := #DSI, DataIn :=, Cin :=, Config := #Config.Vrt_1, Alarm := #Alarm.Vrt_1, Warning := #Warning.Vrt_1, MachineInterface =>, COut => #COut.Vrt_1, DataOut =>)
   END_RUNG
   // the same network as SCL:
   #Vrt_1(AreaInterface := #AreaInterface,   // "ValveMachine_FB"
          ZSI := #ZSI,
          DSI := #DSI,
          Config := #Config.Vrt_1,
          Alarm := #Alarm.Vrt_1,
          Warning := #Warning.Vrt_1,
          COut => #COut.Vrt_1);
END_REGION

REGION Network 28: Verticale_2 - Valve Manager
   RUNG wire#powerrail
      #Vrt_2(AreaInterface := #AreaInterface, ZSI := #ZSI, DSI := #DSI, DataIn :=, Cin :=, Config := #Config.Vrt_2, Alarm := #Alarm.Vrt_2, Warning := #Warning.Vrt_2, MachineInterface =>, COut => #COut.Vrt_2, DataOut =>)
   END_RUNG
   // the same network as SCL:
   #Vrt_2(AreaInterface := #AreaInterface,   // "ValveMachine_FB"
          ZSI := #ZSI,
          DSI := #DSI,
          Config := #Config.Vrt_2,
          Alarm := #Alarm.Vrt_2,
          Warning := #Warning.Vrt_2,
          COut => #COut.Vrt_2);
END_REGION

REGION Network 29: << GESTIONE ORIZZONTALE >>
END_REGION

REGION Network 30: <+>
END_REGION

REGION Network 31: << GESTIONE SPINTORE ORIZZ_1&2 - ANALOGIC SENSOR >>
END_REGION

REGION Network 33: Orizzontale_1 -Scalatura sensore
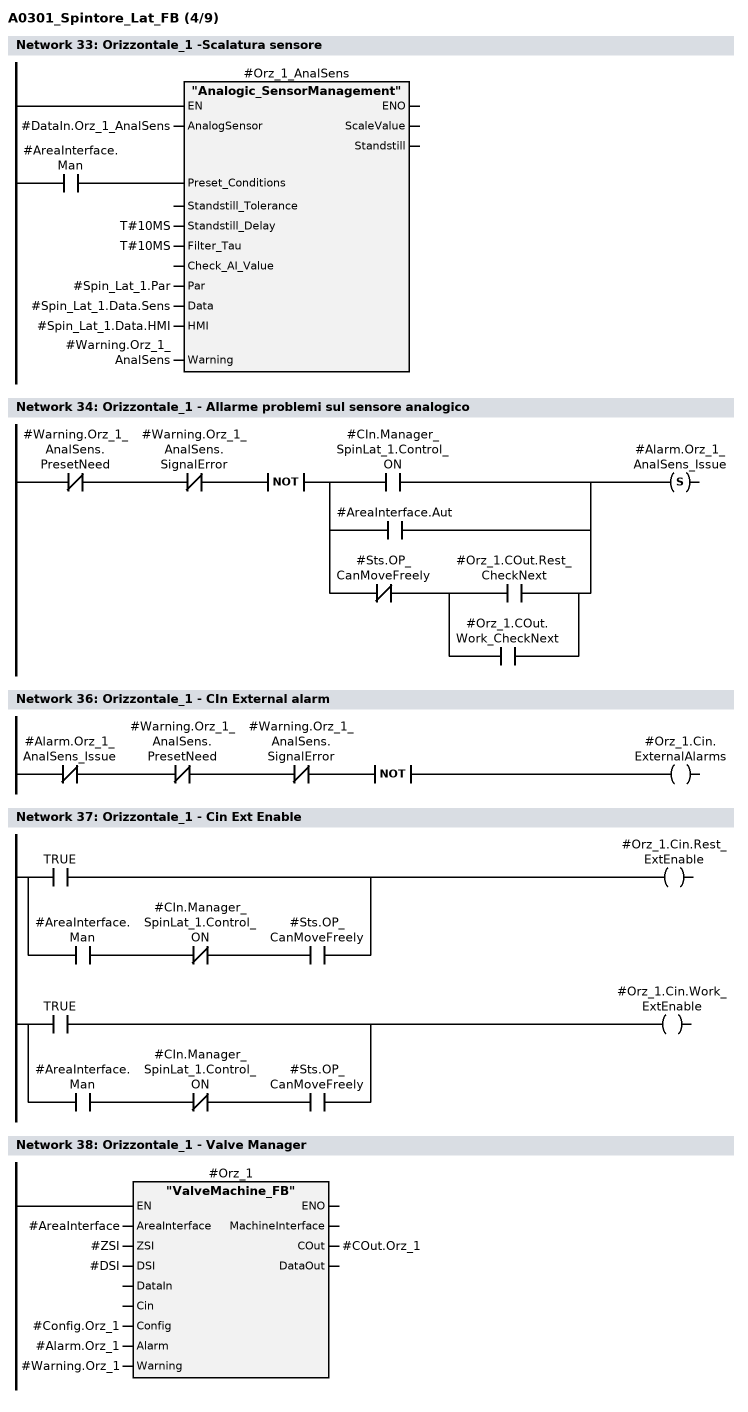
   RUNG wire#powerrail
      #Orz_1_AnalSens(Preset_Conditions := wire#w1, AnalogSensor := #DataIn.Orz_1_AnalSens, Standstill_Tolerance :=, Standstill_Delay := T#10MS, Filter_Tau := T#10MS, Check_AI_Value :=, Par := #Spin_Lat_1.Par, Data := #Spin_Lat_1.Data.Sens, HMI := #Spin_Lat_1.Data.HMI, Warning := #Warning.Orz_1_AnalSens, ScaleValue =>, Standstill =>)
   END_RUNG
   RUNG wire#powerrail
      Contact( #AreaInterface.Man )
   END_RUNG wire#w1
   // the same network as SCL:
   #Orz_1_AnalSens(AnalogSensor := #DataIn.Orz_1_AnalSens,   // "Analogic_SensorManagement"
                   Preset_Conditions := #AreaInterface.Man,
                   Standstill_Delay := T#10MS,
                   Filter_Tau := T#10MS,
                   Par := #Spin_Lat_1.Par,
                   Data := #Spin_Lat_1.Data.Sens,
                   HMI := #Spin_Lat_1.Data.HMI,
                   Warning := #Warning.Orz_1_AnalSens);
END_REGION

REGION Network 34: Orizzontale_1 - Allarme problemi sul sensore analogico
   RUNG wire#powerrail
      I_Contact( #Warning.Orz_1_AnalSens.PresetNeed )
      I_Contact( #Warning.Orz_1_AnalSens.SignalError )
      Not()
      wire#w1
      Contact( #CIn.Manager_SpinLat_1.Control_ON )
      wire#w2
      S_Coil( #Alarm.Orz_1_AnalSens_Issue )
   END_RUNG
   RUNG wire#w1
      Contact( #AreaInterface.Aut )
   END_RUNG wire#w2
   RUNG wire#w1
      I_Contact( #Sts.OP_CanMoveFreely )
      wire#w3
      Contact( #Orz_1.COut.Rest_CheckNext )
   END_RUNG wire#w2
   RUNG wire#w3
      Contact( #Orz_1.COut.Work_CheckNext )
   END_RUNG wire#w2
   // the same network as SCL:
   IF NOT (NOT #Warning.Orz_1_AnalSens.PresetNeed AND NOT #Warning.Orz_1_AnalSens.SignalError) AND (#CIn.Manager_SpinLat_1.Control_ON OR #AreaInterface.Aut OR (NOT #Sts.OP_CanMoveFreely AND (#Orz_1.COut.Rest_CheckNext OR #Orz_1.COut.Work_CheckNext))) THEN
       #Alarm.Orz_1_AnalSens_Issue := TRUE;
   END_IF;
END_REGION

REGION Network 35 (SCL): Orizzontale_1 - Datain / Config
   // DataIn Scritti sulla CALL dell'FB

   #Orz_1.Config := #Config.Orz_1;

   IF #Spin_Lat_1.Par.Enable AND #Sts.Beam.H_B > 0.0 THEN

       #Orz_1.DataIn.Work_Ls[1] := #Vrt_1.DataIn.Work_Ls[1] := ABS (#Orz_1_AnalSens.ScaleValue - #Sts.Beam.H_B) <= #Spin_Lat_1.Par_Mach.Tol_Work;
       #Orz_1.Config.V.WorkLimSwitchExist := TRUE;
       #Orz_1.Config.V.WorkTime := T#0.01s;

   ELSIF #Ctrl.OP_Rest THEN
       #Orz_1.DataIn.Work_Ls[1] := FALSE;
       #Vrt_1.DataIn.Work_Ls[1] := FALSE;

       // ********************************************************************************************************************************************
   ELSE
       // Overide della configurazione di default della valvola

       #Orz_1.Config.V.WorkLimSwitchExist := FALSE;
       #Orz_1.Config.V.WorkTime := #Spin_Lat_1.Par_Mach.WorkTime_SensDisable;
   END_IF;
END_REGION

REGION Network 36: Orizzontale_1 - CIn External alarm
   RUNG wire#powerrail
      I_Contact( #Alarm.Orz_1_AnalSens_Issue )
      I_Contact( #Warning.Orz_1_AnalSens.PresetNeed )
      I_Contact( #Warning.Orz_1_AnalSens.SignalError )
      Not()
      Coil( #Orz_1.Cin.ExternalAlarms )
   END_RUNG
   // the same network as SCL:
   #Orz_1.Cin.ExternalAlarms := NOT (NOT #Alarm.Orz_1_AnalSens_Issue AND NOT #Warning.Orz_1_AnalSens.PresetNeed AND NOT #Warning.Orz_1_AnalSens.SignalError);
END_REGION

REGION Network 37: Orizzontale_1 - Cin Ext Enable
   RUNG wire#powerrail
      Contact( TRUE )
      wire#w1
      Coil( #Orz_1.Cin.Rest_ExtEnable )
   END_RUNG
   RUNG wire#powerrail
      Contact( #AreaInterface.Man )
      I_Contact( #CIn.Manager_SpinLat_1.Control_ON )
      Contact( #Sts.OP_CanMoveFreely )
   END_RUNG wire#w1
   RUNG wire#powerrail
      Contact( TRUE )
      wire#w2
      Coil( #Orz_1.Cin.Work_ExtEnable )
   END_RUNG
   RUNG wire#powerrail
      Contact( #AreaInterface.Man )
      I_Contact( #CIn.Manager_SpinLat_1.Control_ON )
      Contact( #Sts.OP_CanMoveFreely )
   END_RUNG wire#w2
   // the same network as SCL:
   #Orz_1.Cin.Rest_ExtEnable := TRUE OR (#AreaInterface.Man AND NOT #CIn.Manager_SpinLat_1.Control_ON AND #Sts.OP_CanMoveFreely);
   #Orz_1.Cin.Work_ExtEnable := TRUE OR (#AreaInterface.Man AND NOT #CIn.Manager_SpinLat_1.Control_ON AND #Sts.OP_CanMoveFreely);
END_REGION

REGION Network 38: Orizzontale_1 - Valve Manager
   RUNG wire#powerrail
      #Orz_1(AreaInterface := #AreaInterface, ZSI := #ZSI, DSI := #DSI, DataIn :=, Cin :=, Config := #Config.Orz_1, Alarm := #Alarm.Orz_1, Warning := #Warning.Orz_1, MachineInterface =>, COut => #COut.Orz_1, DataOut =>)
   END_RUNG
   // the same network as SCL:
   #Orz_1(AreaInterface := #AreaInterface,   // "ValveMachine_FB"
          ZSI := #ZSI,
          DSI := #DSI,
          Config := #Config.Orz_1,
          Alarm := #Alarm.Orz_1,
          Warning := #Warning.Orz_1,
          COut => #COut.Orz_1);
END_REGION

REGION Network 39: <+>
END_REGION

REGION Network 40: Orizzontale_2 -Scalatura sensore
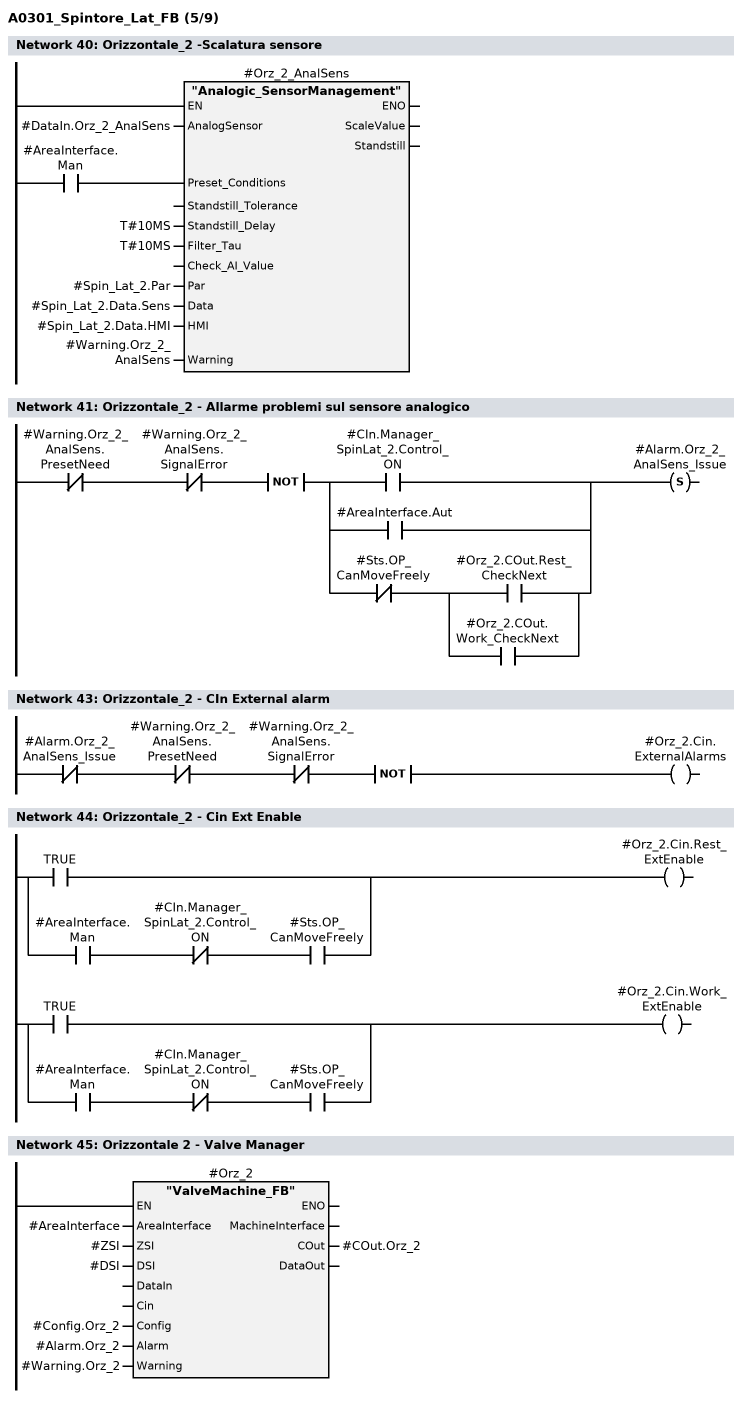
   RUNG wire#powerrail
      #Orz_2_AnalSens(Preset_Conditions := wire#w1, AnalogSensor := #DataIn.Orz_2_AnalSens, Standstill_Tolerance :=, Standstill_Delay := T#10MS, Filter_Tau := T#10MS, Check_AI_Value :=, Par := #Spin_Lat_2.Par, Data := #Spin_Lat_2.Data.Sens, HMI := #Spin_Lat_2.Data.HMI, Warning := #Warning.Orz_2_AnalSens, ScaleValue =>, Standstill =>)
   END_RUNG
   RUNG wire#powerrail
      Contact( #AreaInterface.Man )
   END_RUNG wire#w1
   // the same network as SCL:
   #Orz_2_AnalSens(AnalogSensor := #DataIn.Orz_2_AnalSens,   // "Analogic_SensorManagement"
                   Preset_Conditions := #AreaInterface.Man,
                   Standstill_Delay := T#10MS,
                   Filter_Tau := T#10MS,
                   Par := #Spin_Lat_2.Par,
                   Data := #Spin_Lat_2.Data.Sens,
                   HMI := #Spin_Lat_2.Data.HMI,
                   Warning := #Warning.Orz_2_AnalSens);
END_REGION

REGION Network 41: Orizzontale_2 - Allarme problemi sul sensore analogico
   RUNG wire#powerrail
      I_Contact( #Warning.Orz_2_AnalSens.PresetNeed )
      I_Contact( #Warning.Orz_2_AnalSens.SignalError )
      Not()
      wire#w1
      Contact( #CIn.Manager_SpinLat_2.Control_ON )
      wire#w2
      S_Coil( #Alarm.Orz_2_AnalSens_Issue )
   END_RUNG
   RUNG wire#w1
      Contact( #AreaInterface.Aut )
   END_RUNG wire#w2
   RUNG wire#w1
      I_Contact( #Sts.OP_CanMoveFreely )
      wire#w3
      Contact( #Orz_2.COut.Rest_CheckNext )
   END_RUNG wire#w2
   RUNG wire#w3
      Contact( #Orz_2.COut.Work_CheckNext )
   END_RUNG wire#w2
   // the same network as SCL:
   IF NOT (NOT #Warning.Orz_2_AnalSens.PresetNeed AND NOT #Warning.Orz_2_AnalSens.SignalError) AND (#CIn.Manager_SpinLat_2.Control_ON OR #AreaInterface.Aut OR (NOT #Sts.OP_CanMoveFreely AND (#Orz_2.COut.Rest_CheckNext OR #Orz_2.COut.Work_CheckNext))) THEN
       #Alarm.Orz_2_AnalSens_Issue := TRUE;
   END_IF;
END_REGION

REGION Network 42 (SCL): Orizzontale_2 - Datain / Config
   // DataIn Scritti sulla CALL dell'FB
   #Orz_2.Config := #Config.Orz_2;
   #Spin_Lat_2.Par.Enable := TRUE;

   // Se dal controllo di misura la lunghezza del Beam supera la Quota di abilitazione Spintore 2 abilito il controllo del sensore compensatore sul cilindro ORZ
   IF #Sts."En/Dis_SpinLat_2" THEN

   // *******************************************************************************************************************
   IF  #Spin_Lat_2.Par.Enable AND #Sts.Beam.H_B > 0.0 THEN
       #Spin_Lat_2.Par_Mach.Tol_Work := #Spin_Lat_1.Par_Mach.Tol_Work;

       #Orz_2.DataIn.Work_Ls[1] := #Vrt_2.DataIn.Work_Ls[1] := ABS (#Orz_2_AnalSens.ScaleValue - #Sts.Beam.H_B) <= #Spin_Lat_2.Par_Mach.Tol_Work;
       #Orz_2.Config.V.WorkLimSwitchExist := TRUE;
       #Orz_2.Config.V.WorkTime := T#0.01s;

   ELSIF #Ctrl.OP_Rest THEN
       #Orz_2.DataIn.Work_Ls[1] := FALSE;
       #Vrt_2.DataIn.Work_Ls[1] := FALSE;

       // ***************************************************************************************************************
   ELSE
       // Overide della configurazione di default della valvola

       #Orz_2.DataIn.Work_Ls[1] := FALSE;
       #Orz_2.Config.V.WorkLimSwitchExist := FALSE;
       #Orz_2.Config.V.WorkTime := #Spin_Lat_2.Par_Mach.WorkTime_SensDisable;
   END_IF;
   END_IF;
END_REGION

REGION Network 43: Orizzontale_2 - CIn External alarm
   RUNG wire#powerrail
      I_Contact( #Alarm.Orz_2_AnalSens_Issue )
      I_Contact( #Warning.Orz_2_AnalSens.PresetNeed )
      I_Contact( #Warning.Orz_2_AnalSens.SignalError )
      Not()
      Coil( #Orz_2.Cin.ExternalAlarms )
   END_RUNG
   // the same network as SCL:
   #Orz_2.Cin.ExternalAlarms := NOT (NOT #Alarm.Orz_2_AnalSens_Issue AND NOT #Warning.Orz_2_AnalSens.PresetNeed AND NOT #Warning.Orz_2_AnalSens.SignalError);
END_REGION

REGION Network 44: Orizzontale_2 - Cin Ext Enable
   RUNG wire#powerrail
      Contact( TRUE )
      wire#w1
      Coil( #Orz_2.Cin.Rest_ExtEnable )
   END_RUNG
   RUNG wire#powerrail
      Contact( #AreaInterface.Man )
      I_Contact( #CIn.Manager_SpinLat_2.Control_ON )
      Contact( #Sts.OP_CanMoveFreely )
   END_RUNG wire#w1
   RUNG wire#powerrail
      Contact( TRUE )
      wire#w2
      Coil( #Orz_2.Cin.Work_ExtEnable )
   END_RUNG
   RUNG wire#powerrail
      Contact( #AreaInterface.Man )
      I_Contact( #CIn.Manager_SpinLat_2.Control_ON )
      Contact( #Sts.OP_CanMoveFreely )
   END_RUNG wire#w2
   // the same network as SCL:
   #Orz_2.Cin.Rest_ExtEnable := TRUE OR (#AreaInterface.Man AND NOT #CIn.Manager_SpinLat_2.Control_ON AND #Sts.OP_CanMoveFreely);
   #Orz_2.Cin.Work_ExtEnable := TRUE OR (#AreaInterface.Man AND NOT #CIn.Manager_SpinLat_2.Control_ON AND #Sts.OP_CanMoveFreely);
END_REGION

REGION Network 45: Orizzontale 2 - Valve Manager
   RUNG wire#powerrail
      #Orz_2(AreaInterface := #AreaInterface, ZSI := #ZSI, DSI := #DSI, DataIn :=, Cin :=, Config := #Config.Orz_2, Alarm := #Alarm.Orz_2, Warning := #Warning.Orz_2, MachineInterface =>, COut => #COut.Orz_2, DataOut =>)
   END_RUNG
   // the same network as SCL:
   #Orz_2(AreaInterface := #AreaInterface,   // "ValveMachine_FB"
          ZSI := #ZSI,
          DSI := #DSI,
          Config := #Config.Orz_2,
          Alarm := #Alarm.Orz_2,
          Warning := #Warning.Orz_2,
          COut => #COut.Orz_2);
END_REGION

REGION Network 47: << GESTIONE SOLLEVATORI >>
END_REGION

REGION Network 48: S[1...6] Sollevatori - CIn External alarm
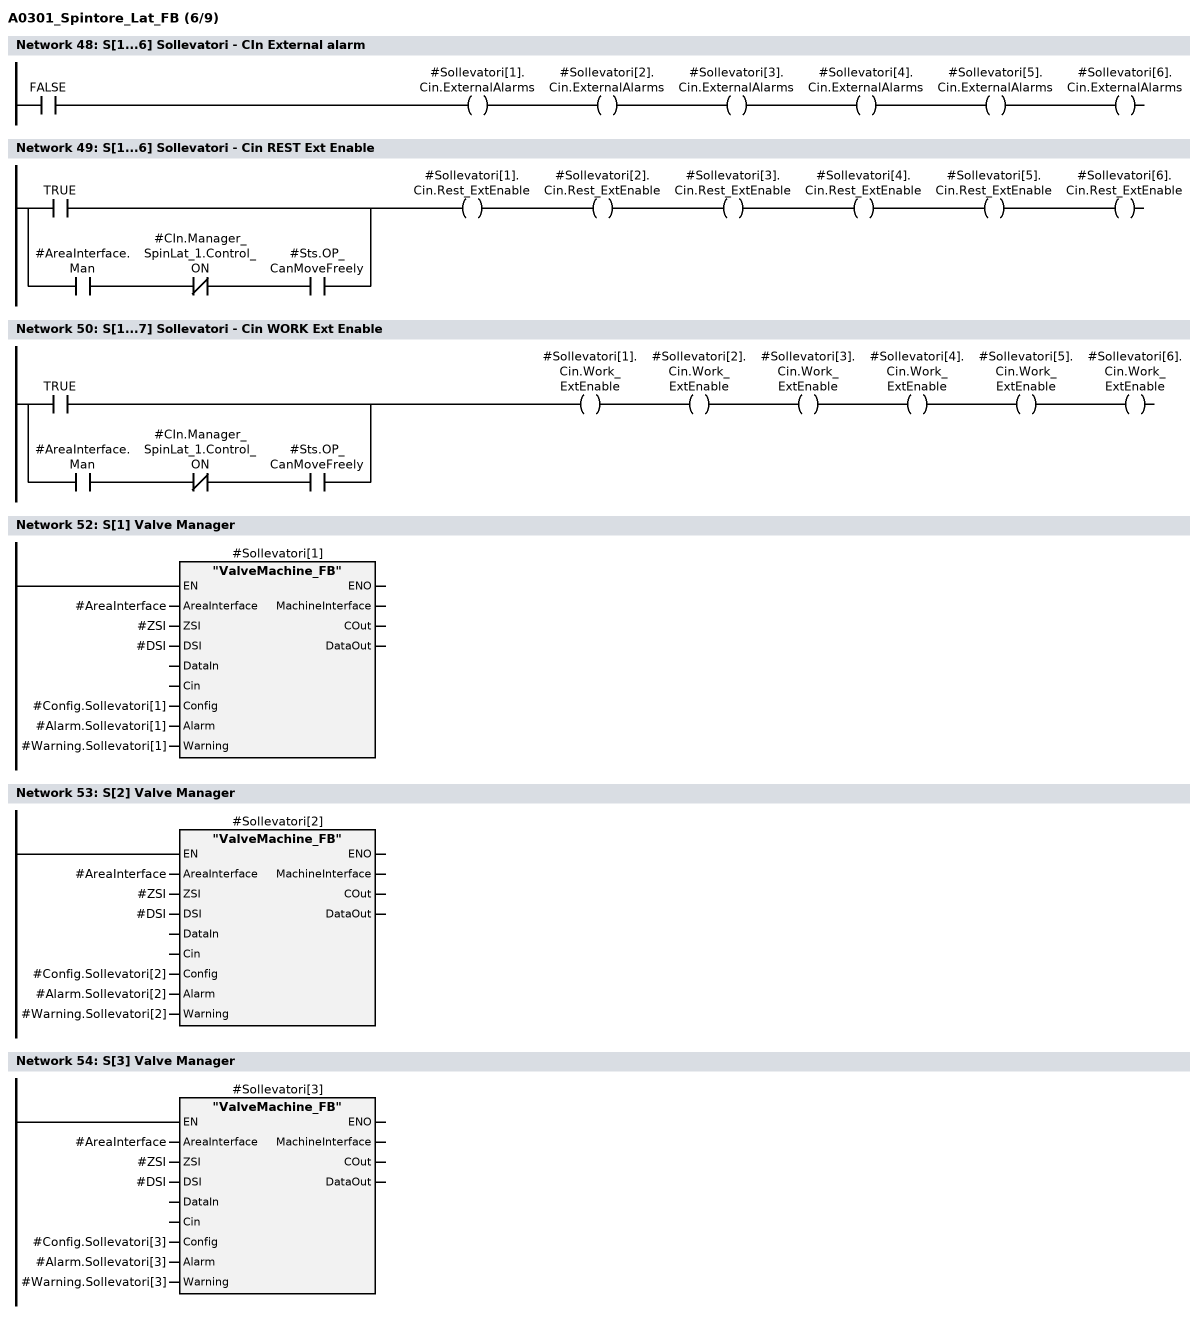
   RUNG wire#powerrail
      Contact( FALSE )
      Coil( #Sollevatori[1].Cin.ExternalAlarms )
      Coil( #Sollevatori[2].Cin.ExternalAlarms )
      Coil( #Sollevatori[3].Cin.ExternalAlarms )
      Coil( #Sollevatori[4].Cin.ExternalAlarms )
      Coil( #Sollevatori[5].Cin.ExternalAlarms )
      Coil( #Sollevatori[6].Cin.ExternalAlarms )
   END_RUNG
   // the same network as SCL:
   #Sollevatori[1].Cin.ExternalAlarms := FALSE;
   #Sollevatori[2].Cin.ExternalAlarms := FALSE;
   #Sollevatori[3].Cin.ExternalAlarms := FALSE;
   #Sollevatori[4].Cin.ExternalAlarms := FALSE;
   #Sollevatori[5].Cin.ExternalAlarms := FALSE;
   #Sollevatori[6].Cin.ExternalAlarms := FALSE;
END_REGION

REGION Network 49: S[1...6] Sollevatori - Cin REST Ext Enable
   RUNG wire#powerrail
      Contact( TRUE )
      wire#w1
      Coil( #Sollevatori[1].Cin.Rest_ExtEnable )
      Coil( #Sollevatori[2].Cin.Rest_ExtEnable )
      Coil( #Sollevatori[3].Cin.Rest_ExtEnable )
      Coil( #Sollevatori[4].Cin.Rest_ExtEnable )
      Coil( #Sollevatori[5].Cin.Rest_ExtEnable )
      Coil( #Sollevatori[6].Cin.Rest_ExtEnable )
   END_RUNG
   RUNG wire#powerrail
      Contact( #AreaInterface.Man )
      I_Contact( #CIn.Manager_SpinLat_1.Control_ON )
      Contact( #Sts.OP_CanMoveFreely )
   END_RUNG wire#w1
   // the same network as SCL:
   #Sollevatori[1].Cin.Rest_ExtEnable := TRUE OR (#AreaInterface.Man AND NOT #CIn.Manager_SpinLat_1.Control_ON AND #Sts.OP_CanMoveFreely);
   #Sollevatori[2].Cin.Rest_ExtEnable := TRUE OR (#AreaInterface.Man AND NOT #CIn.Manager_SpinLat_1.Control_ON AND #Sts.OP_CanMoveFreely);
   #Sollevatori[3].Cin.Rest_ExtEnable := TRUE OR (#AreaInterface.Man AND NOT #CIn.Manager_SpinLat_1.Control_ON AND #Sts.OP_CanMoveFreely);
   #Sollevatori[4].Cin.Rest_ExtEnable := TRUE OR (#AreaInterface.Man AND NOT #CIn.Manager_SpinLat_1.Control_ON AND #Sts.OP_CanMoveFreely);
   #Sollevatori[5].Cin.Rest_ExtEnable := TRUE OR (#AreaInterface.Man AND NOT #CIn.Manager_SpinLat_1.Control_ON AND #Sts.OP_CanMoveFreely);
   #Sollevatori[6].Cin.Rest_ExtEnable := TRUE OR (#AreaInterface.Man AND NOT #CIn.Manager_SpinLat_1.Control_ON AND #Sts.OP_CanMoveFreely);
END_REGION

REGION Network 50: S[1...7] Sollevatori - Cin WORK Ext Enable
   RUNG wire#powerrail
      Contact( TRUE )
      wire#w1
      Coil( #Sollevatori[1].Cin.Work_ExtEnable )
      Coil( #Sollevatori[2].Cin.Work_ExtEnable )
      Coil( #Sollevatori[3].Cin.Work_ExtEnable )
      Coil( #Sollevatori[4].Cin.Work_ExtEnable )
      Coil( #Sollevatori[5].Cin.Work_ExtEnable )
      Coil( #Sollevatori[6].Cin.Work_ExtEnable )
   END_RUNG
   RUNG wire#powerrail
      Contact( #AreaInterface.Man )
      I_Contact( #CIn.Manager_SpinLat_1.Control_ON )
      Contact( #Sts.OP_CanMoveFreely )
   END_RUNG wire#w1
   // the same network as SCL:
   #Sollevatori[1].Cin.Work_ExtEnable := TRUE OR (#AreaInterface.Man AND NOT #CIn.Manager_SpinLat_1.Control_ON AND #Sts.OP_CanMoveFreely);
   #Sollevatori[2].Cin.Work_ExtEnable := TRUE OR (#AreaInterface.Man AND NOT #CIn.Manager_SpinLat_1.Control_ON AND #Sts.OP_CanMoveFreely);
   #Sollevatori[3].Cin.Work_ExtEnable := TRUE OR (#AreaInterface.Man AND NOT #CIn.Manager_SpinLat_1.Control_ON AND #Sts.OP_CanMoveFreely);
   #Sollevatori[4].Cin.Work_ExtEnable := TRUE OR (#AreaInterface.Man AND NOT #CIn.Manager_SpinLat_1.Control_ON AND #Sts.OP_CanMoveFreely);
   #Sollevatori[5].Cin.Work_ExtEnable := TRUE OR (#AreaInterface.Man AND NOT #CIn.Manager_SpinLat_1.Control_ON AND #Sts.OP_CanMoveFreely);
   #Sollevatori[6].Cin.Work_ExtEnable := TRUE OR (#AreaInterface.Man AND NOT #CIn.Manager_SpinLat_1.Control_ON AND #Sts.OP_CanMoveFreely);
END_REGION

REGION Network 51: <+>
END_REGION

REGION Network 52: S[1] Valve Manager
   RUNG wire#powerrail
      #Sollevatori[1](AreaInterface := #AreaInterface, ZSI := #ZSI, DSI := #DSI, DataIn :=, Cin :=, Config := #Config.Sollevatori[1], Alarm := #Alarm.Sollevatori[1], Warning := #Warning.Sollevatori[1], MachineInterface =>, COut =>, DataOut =>)
   END_RUNG
   // the same network as SCL:
   #Sollevatori[1](AreaInterface := #AreaInterface,   // "ValveMachine_FB"
                   ZSI := #ZSI,
                   DSI := #DSI,
                   Config := #Config.Sollevatori[1],
                   Alarm := #Alarm.Sollevatori[1],
                   Warning := #Warning.Sollevatori[1]);
END_REGION

REGION Network 53: S[2] Valve Manager
   RUNG wire#powerrail
      #Sollevatori[2](AreaInterface := #AreaInterface, ZSI := #ZSI, DSI := #DSI, DataIn :=, Cin :=, Config := #Config.Sollevatori[2], Alarm := #Alarm.Sollevatori[2], Warning := #Warning.Sollevatori[2], MachineInterface =>, COut =>, DataOut =>)
   END_RUNG
   // the same network as SCL:
   #Sollevatori[2](AreaInterface := #AreaInterface,   // "ValveMachine_FB"
                   ZSI := #ZSI,
                   DSI := #DSI,
                   Config := #Config.Sollevatori[2],
                   Alarm := #Alarm.Sollevatori[2],
                   Warning := #Warning.Sollevatori[2]);
END_REGION

REGION Network 54: S[3] Valve Manager
   RUNG wire#powerrail
      #Sollevatori[3](AreaInterface := #AreaInterface, ZSI := #ZSI, DSI := #DSI, DataIn :=, Cin :=, Config := #Config.Sollevatori[3], Alarm := #Alarm.Sollevatori[3], Warning := #Warning.Sollevatori[3], MachineInterface =>, COut =>, DataOut =>)
   END_RUNG
   // the same network as SCL:
   #Sollevatori[3](AreaInterface := #AreaInterface,   // "ValveMachine_FB"
                   ZSI := #ZSI,
                   DSI := #DSI,
                   Config := #Config.Sollevatori[3],
                   Alarm := #Alarm.Sollevatori[3],
                   Warning := #Warning.Sollevatori[3]);
END_REGION

REGION Network 55: S[4] Valve Manager
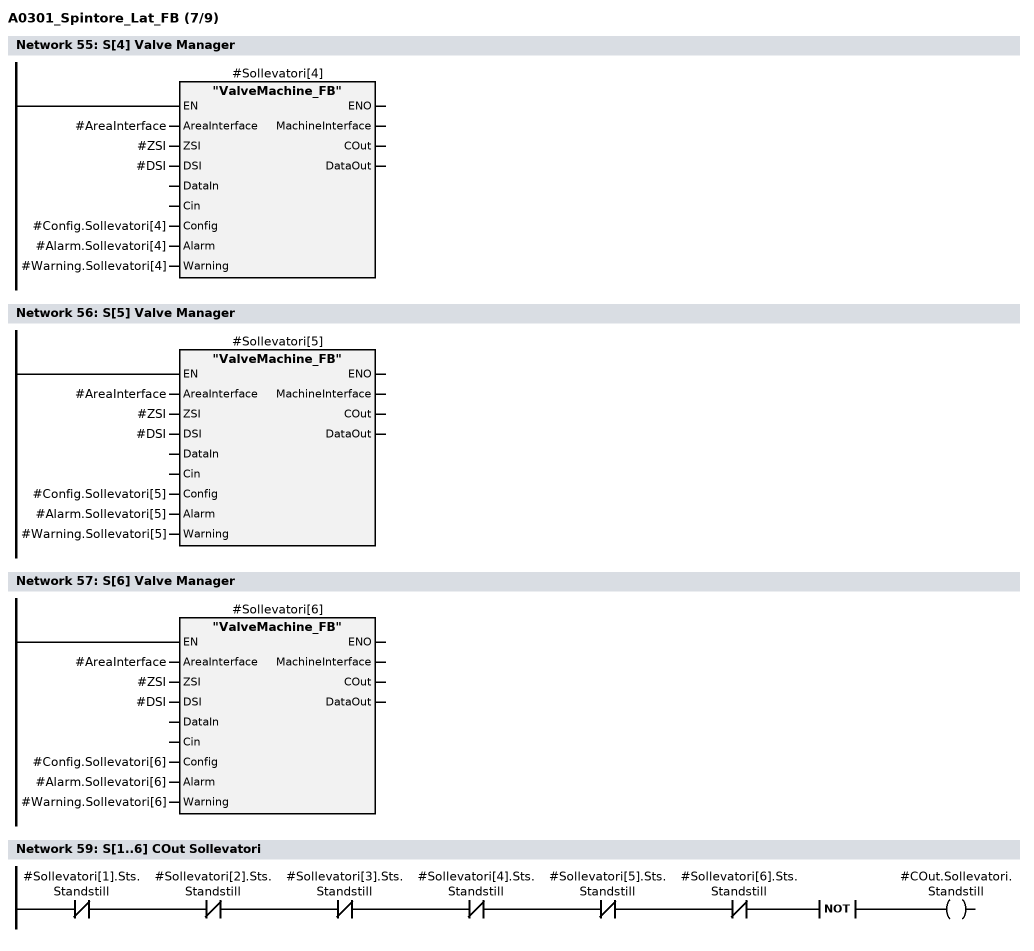
   RUNG wire#powerrail
      #Sollevatori[4](AreaInterface := #AreaInterface, ZSI := #ZSI, DSI := #DSI, DataIn :=, Cin :=, Config := #Config.Sollevatori[4], Alarm := #Alarm.Sollevatori[4], Warning := #Warning.Sollevatori[4], MachineInterface =>, COut =>, DataOut =>)
   END_RUNG
   // the same network as SCL:
   #Sollevatori[4](AreaInterface := #AreaInterface,   // "ValveMachine_FB"
                   ZSI := #ZSI,
                   DSI := #DSI,
                   Config := #Config.Sollevatori[4],
                   Alarm := #Alarm.Sollevatori[4],
                   Warning := #Warning.Sollevatori[4]);
END_REGION

REGION Network 56: S[5] Valve Manager
   RUNG wire#powerrail
      #Sollevatori[5](AreaInterface := #AreaInterface, ZSI := #ZSI, DSI := #DSI, DataIn :=, Cin :=, Config := #Config.Sollevatori[5], Alarm := #Alarm.Sollevatori[5], Warning := #Warning.Sollevatori[5], MachineInterface =>, COut =>, DataOut =>)
   END_RUNG
   // the same network as SCL:
   #Sollevatori[5](AreaInterface := #AreaInterface,   // "ValveMachine_FB"
                   ZSI := #ZSI,
                   DSI := #DSI,
                   Config := #Config.Sollevatori[5],
                   Alarm := #Alarm.Sollevatori[5],
                   Warning := #Warning.Sollevatori[5]);
END_REGION

REGION Network 57: S[6] Valve Manager
   RUNG wire#powerrail
      #Sollevatori[6](AreaInterface := #AreaInterface, ZSI := #ZSI, DSI := #DSI, DataIn :=, Cin :=, Config := #Config.Sollevatori[6], Alarm := #Alarm.Sollevatori[6], Warning := #Warning.Sollevatori[6], MachineInterface =>, COut =>, DataOut =>)
   END_RUNG
   // the same network as SCL:
   #Sollevatori[6](AreaInterface := #AreaInterface,   // "ValveMachine_FB"
                   ZSI := #ZSI,
                   DSI := #DSI,
                   Config := #Config.Sollevatori[6],
                   Alarm := #Alarm.Sollevatori[6],
                   Warning := #Warning.Sollevatori[6]);
END_REGION

REGION Network 58: <+>
END_REGION

REGION Network 59: S[1..6] COut Sollevatori
   RUNG wire#powerrail
      I_Contact( #Sollevatori[1].Sts.Standstill )
      I_Contact( #Sollevatori[2].Sts.Standstill )
      I_Contact( #Sollevatori[3].Sts.Standstill )
      I_Contact( #Sollevatori[4].Sts.Standstill )
      I_Contact( #Sollevatori[5].Sts.Standstill )
      I_Contact( #Sollevatori[6].Sts.Standstill )
      Not()
      Coil( #COut.Sollevatori.Standstill )
   END_RUNG
   // the same network as SCL:
   #COut.Sollevatori.Standstill := NOT (NOT #Sollevatori[1].Sts.Standstill AND NOT #Sollevatori[2].Sts.Standstill AND NOT #Sollevatori[3].Sts.Standstill AND NOT #Sollevatori[4].Sts.Standstill AND NOT #Sollevatori[5].Sts.Standstill AND NOT #Sollevatori[6].Sts.Standstill);
END_REGION

REGION Network 60 (SCL): S[1..6] COut Sollevatori


   // Controllo uscita COut AT_REST in base allo stato di tutti i Sollevatori
   IF  #Sollevatori[1].COut.Rest AND
       #Sollevatori[2].COut.Rest AND
       #Sollevatori[3].COut.Rest AND
       #Sollevatori[4].COut.Rest AND
       #Sollevatori[5].COut.Rest AND
       #Sollevatori[6].COut.Rest THEN
       #COut.Sollevatori.Rest := 1;
   ELSE
       #COut.Sollevatori.Rest := 0;
   END_IF;

   // Controllo uscita COut AT_WORK in base allo stato di tutti i Sollevatori
   IF  #Sollevatori[1].COut.Work AND
       #Sollevatori[2].COut.Work AND
       #Sollevatori[3].COut.Work AND
       #Sollevatori[4].COut.Work AND
       #Sollevatori[5].COut.Work AND
       #Sollevatori[6].COut.Work THEN
       #COut.Sollevatori.Work := 1;
   ELSE
       #COut.Sollevatori.Work := 0;
   END_IF;
END_REGION

REGION Network 61: <+>
END_REGION

REGION Network 62: Stazione COut
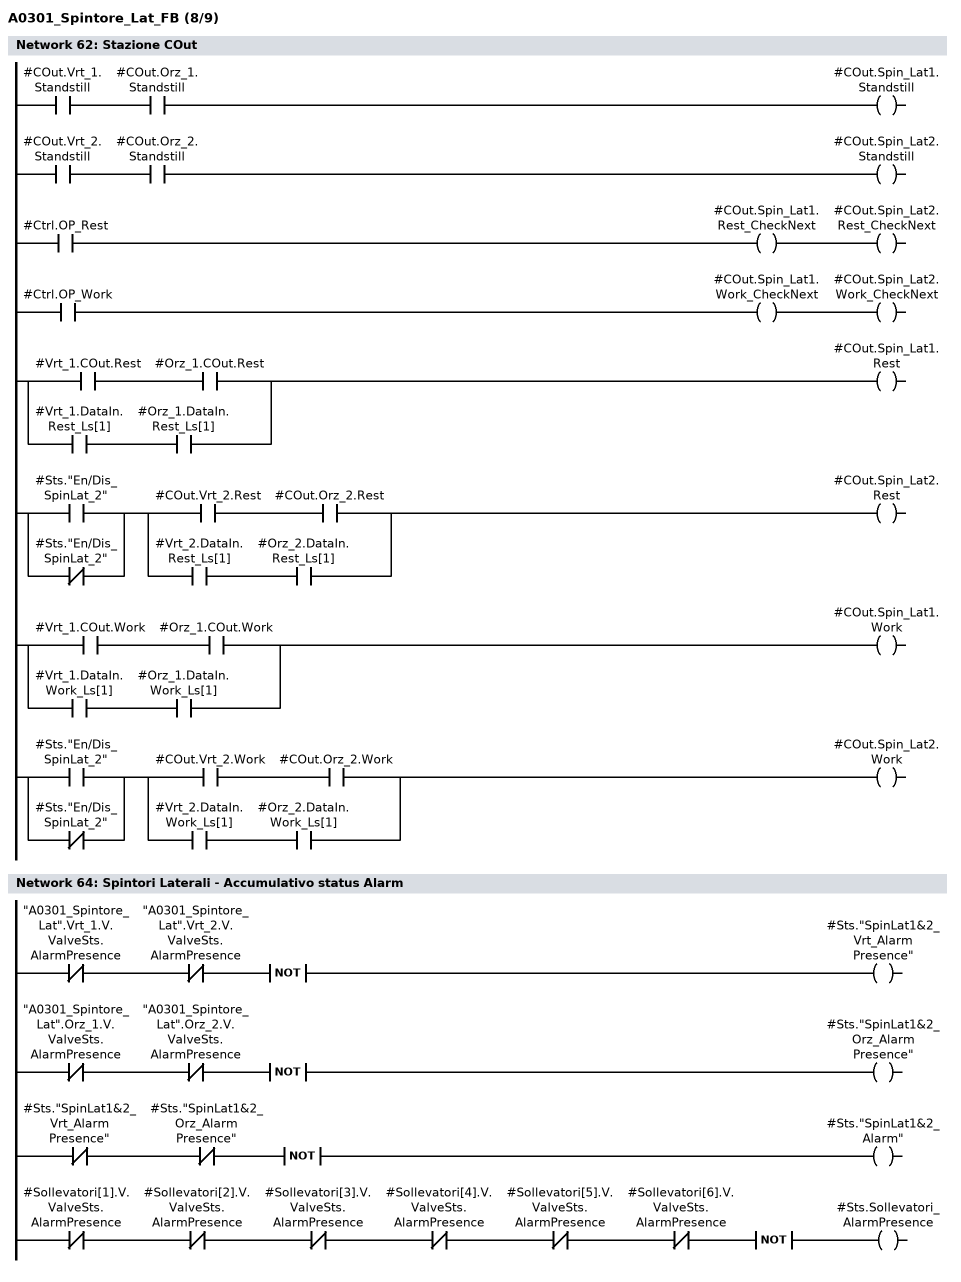
   RUNG wire#powerrail
      Contact( #COut.Vrt_1.Standstill )
      Contact( #COut.Orz_1.Standstill )
      Coil( #COut.Spin_Lat1.Standstill )
   END_RUNG
   RUNG wire#powerrail
      Contact( #COut.Vrt_2.Standstill )
      Contact( #COut.Orz_2.Standstill )
      Coil( #COut.Spin_Lat2.Standstill )
   END_RUNG
   RUNG wire#powerrail
      Contact( #Ctrl.OP_Rest )
      Coil( #COut.Spin_Lat1.Rest_CheckNext )
      Coil( #COut.Spin_Lat2.Rest_CheckNext )
   END_RUNG
   RUNG wire#powerrail
      Contact( #Ctrl.OP_Work )
      Coil( #COut.Spin_Lat1.Work_CheckNext )
      Coil( #COut.Spin_Lat2.Work_CheckNext )
   END_RUNG
   RUNG wire#powerrail
      Contact( #Vrt_1.COut.Rest )
      Contact( #Orz_1.COut.Rest )
      wire#w1
      Coil( #COut.Spin_Lat1.Rest )
   END_RUNG
   RUNG wire#powerrail
      Contact( #Vrt_1.DataIn.Rest_Ls[1] )
      Contact( #Orz_1.DataIn.Rest_Ls[1] )
   END_RUNG wire#w1
   RUNG wire#powerrail
      Contact( #Sts."En/Dis_SpinLat_2" )
      wire#w2
      Contact( #COut.Vrt_2.Rest )
      Contact( #COut.Orz_2.Rest )
      wire#w3
      Coil( #COut.Spin_Lat2.Rest )
   END_RUNG
   RUNG wire#powerrail
      I_Contact( #Sts."En/Dis_SpinLat_2" )
   END_RUNG wire#w2
   RUNG wire#w2
      Contact( #Vrt_2.DataIn.Rest_Ls[1] )
      Contact( #Orz_2.DataIn.Rest_Ls[1] )
   END_RUNG wire#w3
   RUNG wire#powerrail
      Contact( #Vrt_1.COut.Work )
      Contact( #Orz_1.COut.Work )
      wire#w4
      Coil( #COut.Spin_Lat1.Work )
   END_RUNG
   RUNG wire#powerrail
      Contact( #Vrt_1.DataIn.Work_Ls[1] )
      Contact( #Orz_1.DataIn.Work_Ls[1] )
   END_RUNG wire#w4
   RUNG wire#powerrail
      Contact( #Sts."En/Dis_SpinLat_2" )
      wire#w5
      Contact( #COut.Vrt_2.Work )
      Contact( #COut.Orz_2.Work )
      wire#w6
      Coil( #COut.Spin_Lat2.Work )
   END_RUNG
   RUNG wire#powerrail
      I_Contact( #Sts."En/Dis_SpinLat_2" )
   END_RUNG wire#w5
   RUNG wire#w5
      Contact( #Vrt_2.DataIn.Work_Ls[1] )
      Contact( #Orz_2.DataIn.Work_Ls[1] )
   END_RUNG wire#w6
   // the same network as SCL:
   #COut.Spin_Lat1.Standstill := #COut.Vrt_1.Standstill AND #COut.Orz_1.Standstill;
   #COut.Spin_Lat2.Standstill := #COut.Vrt_2.Standstill AND #COut.Orz_2.Standstill;
   #COut.Spin_Lat1.Rest_CheckNext := #Ctrl.OP_Rest;
   #COut.Spin_Lat2.Rest_CheckNext := #Ctrl.OP_Rest;
   #COut.Spin_Lat1.Work_CheckNext := #Ctrl.OP_Work;
   #COut.Spin_Lat2.Work_CheckNext := #Ctrl.OP_Work;
   #COut.Spin_Lat1.Rest := (#Vrt_1.COut.Rest AND #Orz_1.COut.Rest) OR (#Vrt_1.DataIn.Rest_Ls[1] AND #Orz_1.DataIn.Rest_Ls[1]);
   #COut.Spin_Lat2.Rest := (#Sts."En/Dis_SpinLat_2" OR NOT #Sts."En/Dis_SpinLat_2") AND ((#COut.Vrt_2.Rest AND #COut.Orz_2.Rest) OR (#Vrt_2.DataIn.Rest_Ls[1] AND #Orz_2.DataIn.Rest_Ls[1]));
   #COut.Spin_Lat1.Work := (#Vrt_1.COut.Work AND #Orz_1.COut.Work) OR (#Vrt_1.DataIn.Work_Ls[1] AND #Orz_1.DataIn.Work_Ls[1]);
   #COut.Spin_Lat2.Work := (#Sts."En/Dis_SpinLat_2" OR NOT #Sts."En/Dis_SpinLat_2") AND ((#COut.Vrt_2.Work AND #COut.Orz_2.Work) OR (#Vrt_2.DataIn.Work_Ls[1] AND #Orz_2.DataIn.Work_Ls[1]));
END_REGION

REGION Network 64: Spintori Laterali - Accumulativo status Alarm
   RUNG wire#powerrail
      I_Contact( "A0301_Spintore_Lat".Vrt_1.V.ValveSts.AlarmPresence )
      I_Contact( "A0301_Spintore_Lat".Vrt_2.V.ValveSts.AlarmPresence )
      Not()
      Coil( #Sts."SpinLat1&2_Vrt_AlarmPresence" )
   END_RUNG
   RUNG wire#powerrail
      I_Contact( "A0301_Spintore_Lat".Orz_1.V.ValveSts.AlarmPresence )
      I_Contact( "A0301_Spintore_Lat".Orz_2.V.ValveSts.AlarmPresence )
      Not()
      Coil( #Sts."SpinLat1&2_Orz_AlarmPresence" )
   END_RUNG
   RUNG wire#powerrail
      I_Contact( #Sts."SpinLat1&2_Vrt_AlarmPresence" )
      I_Contact( #Sts."SpinLat1&2_Orz_AlarmPresence" )
      Not()
      Coil( #Sts."SpinLat1&2_Alarm" )
   END_RUNG
   RUNG wire#powerrail
      I_Contact( #Sollevatori[1].V.ValveSts.AlarmPresence )
      I_Contact( #Sollevatori[2].V.ValveSts.AlarmPresence )
      I_Contact( #Sollevatori[3].V.ValveSts.AlarmPresence )
      I_Contact( #Sollevatori[4].V.ValveSts.AlarmPresence )
      I_Contact( #Sollevatori[5].V.ValveSts.AlarmPresence )
      I_Contact( #Sollevatori[6].V.ValveSts.AlarmPresence )
      Not()
      Coil( #Sts.Sollevatori_AlarmPresence )
   END_RUNG
   // the same network as SCL:
   #Sts."SpinLat1&2_Vrt_AlarmPresence" := NOT (NOT "A0301_Spintore_Lat".Vrt_1.V.ValveSts.AlarmPresence AND NOT "A0301_Spintore_Lat".Vrt_2.V.ValveSts.AlarmPresence);
   #Sts."SpinLat1&2_Orz_AlarmPresence" := NOT (NOT "A0301_Spintore_Lat".Orz_1.V.ValveSts.AlarmPresence AND NOT "A0301_Spintore_Lat".Orz_2.V.ValveSts.AlarmPresence);
   #Sts."SpinLat1&2_Alarm" := NOT (NOT #Sts."SpinLat1&2_Vrt_AlarmPresence" AND NOT #Sts."SpinLat1&2_Orz_AlarmPresence");
   #Sts.Sollevatori_AlarmPresence := NOT (NOT #Sollevatori[1].V.ValveSts.AlarmPresence AND NOT #Sollevatori[2].V.ValveSts.AlarmPresence AND NOT #Sollevatori[3].V.ValveSts.AlarmPresence AND NOT #Sollevatori[4].V.ValveSts.AlarmPresence AND NOT #Sollevatori[5].V.ValveSts.AlarmPresence AND NOT #Sollevatori[6].V.ValveSts.AlarmPresence);
END_REGION

REGION Network 65 (SCL): HMI STATUS - Postazione
   // Area dati appoggio per HMI
   // SPINTORE LAT. 1&2 Verticale
   #HMI."SpinLat1&2_Vrt_Sts".Standstill := #COut.Vrt_1.Standstill AND #COut.Vrt_2.Standstill;
   #HMI."SpinLat1&2_Vrt_Sts".Rest := #COut.Vrt_1.Rest AND (#COut.Vrt_2.Rest OR NOT #Sts."En/Dis_SpinLat_2");
   #HMI."SpinLat1&2_Vrt_Sts".Work := #COut.Vrt_1.Work AND (#COut.Vrt_2.Work OR NOT #Sts."En/Dis_SpinLat_2");
   #HMI."SpinLat1&2_Vrt_Sts".AlarmPresence := #Sts."SpinLat1&2_Vrt_AlarmPresence";

   // SPINTORE LAT. 1&2 Orizzontale
   #HMI."SpinLat1&2_Orz_Sts".Standstill := #COut.Orz_1.Standstill AND #COut.Orz_2.Standstill;
   #HMI."SpinLat1&2_Orz_Sts".Rest := #COut.Orz_1.Rest AND (#COut.Orz_2.Rest OR NOT #Sts."En/Dis_SpinLat_2");
   #HMI."SpinLat1&2_Orz_Sts".Work := #COut.Orz_1.Work AND (#COut.Orz_2.Work OR NOT #Sts."En/Dis_SpinLat_2");
   #HMI."SpinLat1&2_Orz_Sts".AlarmPresence := #Sts."SpinLat1&2_Orz_AlarmPresence";

   // Stazione spintori laterati
   #HMI."SpinLat1&2_Sts".Standstill := #COut.Spin_Lat1.Standstill AND (#COut.Spin_Lat2.Standstill OR NOT #Sts."En/Dis_SpinLat_2");
   #HMI."SpinLat1&2_Sts".Rest := #COut.Spin_Lat1.Rest AND (#COut.Spin_Lat2.Rest OR NOT #Sts."En/Dis_SpinLat_2");
   #HMI."SpinLat1&2_Sts".Work := #COut.Spin_Lat1.Work AND(#COut.Spin_Lat2.Work OR NOT #Sts."En/Dis_SpinLat_2");
   #HMI."SpinLat1&2_Sts".AlarmPresence := #Sts."SpinLat1&2_Alarm";

   // Sollevatori
   #HMI.Sollevatori_Sts.Standstill := #COut.Sollevatori.Standstill;
   #HMI.Sollevatori_Sts.Rest := #COut.Sollevatori.Rest;
   #HMI.Sollevatori_Sts.Work := #COut.Sollevatori.Work;
   #HMI.Sollevatori_Sts.AlarmPresence := #Sts.Sollevatori_AlarmPresence;
END_REGION

REGION Network 67: << MAIN MACHINE STATUS >>
END_REGION

REGION Network 68: Machine interface
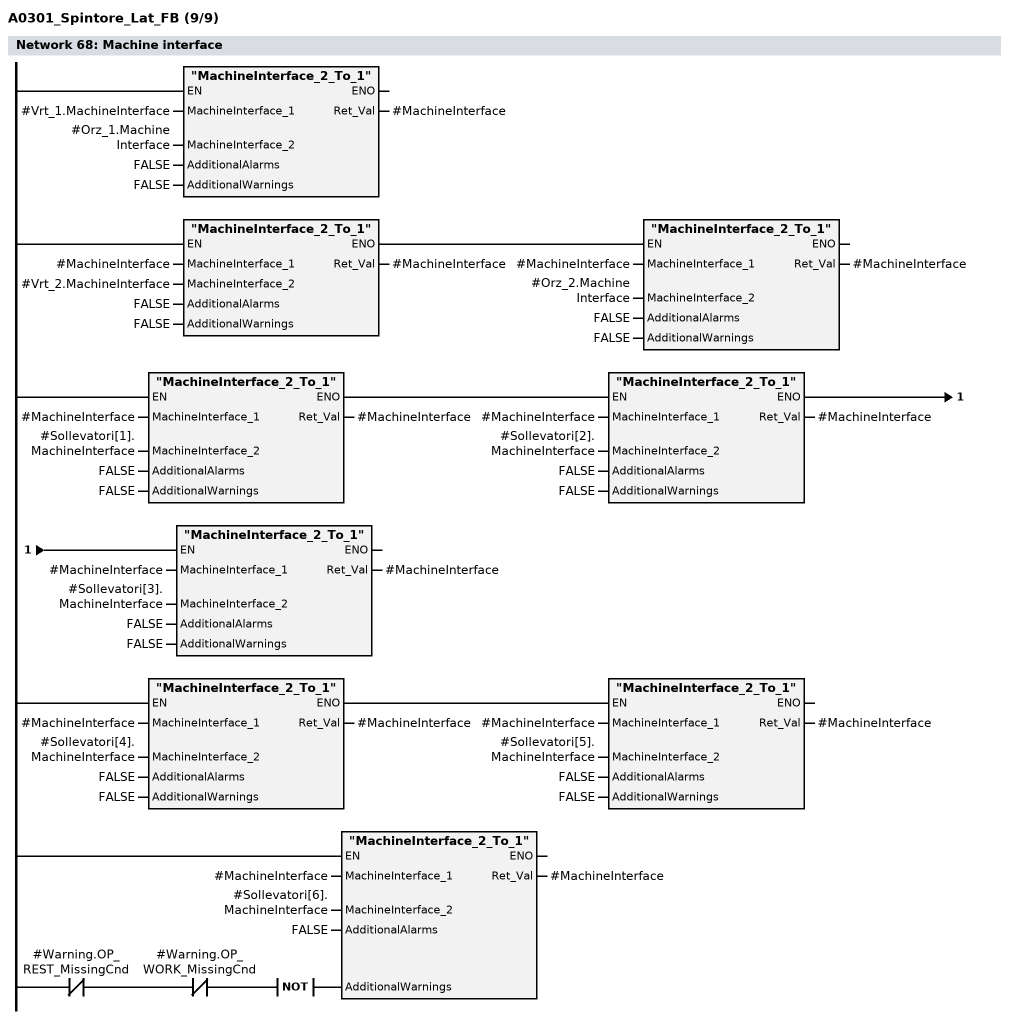
   RUNG wire#powerrail
      "MachineInterface_2_To_1"(MachineInterface_1 := #Vrt_1.MachineInterface, MachineInterface_2 := #Orz_1.MachineInterface, AdditionalAlarms := FALSE, AdditionalWarnings := FALSE, Ret_Val => #MachineInterface)
   END_RUNG
   RUNG wire#powerrail
      "MachineInterface_2_To_1"(MachineInterface_1 := #MachineInterface, MachineInterface_2 := #Vrt_2.MachineInterface, AdditionalAlarms := FALSE, AdditionalWarnings := FALSE, Ret_Val => #MachineInterface)
      "MachineInterface_2_To_1"(MachineInterface_1 := #MachineInterface, MachineInterface_2 := #Orz_2.MachineInterface, AdditionalAlarms := FALSE, AdditionalWarnings := FALSE, Ret_Val => #MachineInterface)
   END_RUNG
   RUNG wire#powerrail
      "MachineInterface_2_To_1"(MachineInterface_1 := #MachineInterface, MachineInterface_2 := #Sollevatori[1].MachineInterface, AdditionalAlarms := FALSE, AdditionalWarnings := FALSE, Ret_Val => #MachineInterface)
      "MachineInterface_2_To_1"(MachineInterface_1 := #MachineInterface, MachineInterface_2 := #Sollevatori[2].MachineInterface, AdditionalAlarms := FALSE, AdditionalWarnings := FALSE, Ret_Val => #MachineInterface)
      "MachineInterface_2_To_1"(MachineInterface_1 := #MachineInterface, MachineInterface_2 := #Sollevatori[3].MachineInterface, AdditionalAlarms := FALSE, AdditionalWarnings := FALSE, Ret_Val => #MachineInterface)
   END_RUNG
   RUNG wire#powerrail
      "MachineInterface_2_To_1"(MachineInterface_1 := #MachineInterface, MachineInterface_2 := #Sollevatori[4].MachineInterface, AdditionalAlarms := FALSE, AdditionalWarnings := FALSE, Ret_Val => #MachineInterface)
      "MachineInterface_2_To_1"(MachineInterface_1 := #MachineInterface, MachineInterface_2 := #Sollevatori[5].MachineInterface, AdditionalAlarms := FALSE, AdditionalWarnings := FALSE, Ret_Val => #MachineInterface)
   END_RUNG
   RUNG wire#powerrail
      "MachineInterface_2_To_1"(AdditionalWarnings := wire#w1, MachineInterface_1 := #MachineInterface, MachineInterface_2 := #Sollevatori[6].MachineInterface, AdditionalAlarms := FALSE, Ret_Val => #MachineInterface)
   END_RUNG
   RUNG wire#powerrail
      I_Contact( #Warning.OP_REST_MissingCnd )
      I_Contact( #Warning.OP_WORK_MissingCnd )
      Not()
   END_RUNG wire#w1
   // the same network as SCL:
   #MachineInterface := "MachineInterface_2_To_1"(MachineInterface_1 := #Vrt_1.MachineInterface,
                           MachineInterface_2 := #Orz_1.MachineInterface,
                           AdditionalAlarms := FALSE,
                           AdditionalWarnings := FALSE);
   #MachineInterface := "MachineInterface_2_To_1"(MachineInterface_1 := #MachineInterface,
                           MachineInterface_2 := #Vrt_2.MachineInterface,
                           AdditionalAlarms := FALSE,
                           AdditionalWarnings := FALSE,
                           ENO => #_w1);
   IF #_w1 THEN
       #MachineInterface := "MachineInterface_2_To_1"(MachineInterface_1 := #MachineInterface,
                               MachineInterface_2 := #Orz_2.MachineInterface,
                               AdditionalAlarms := FALSE,
                               AdditionalWarnings := FALSE);
   END_IF;
   #MachineInterface := "MachineInterface_2_To_1"(MachineInterface_1 := #MachineInterface,
                           MachineInterface_2 := #Sollevatori[1].MachineInterface,
                           AdditionalAlarms := FALSE,
                           AdditionalWarnings := FALSE,
                           ENO => #_w2);
   #MachineInterface := "MachineInterface_2_To_1"(EN := #_w2,
                           MachineInterface_1 := #MachineInterface,
                           MachineInterface_2 := #Sollevatori[2].MachineInterface,
                           AdditionalAlarms := FALSE,
                           AdditionalWarnings := FALSE,
                           ENO => #_w3);
   IF #_w3 THEN
       #MachineInterface := "MachineInterface_2_To_1"(MachineInterface_1 := #MachineInterface,
                               MachineInterface_2 := #Sollevatori[3].MachineInterface,
                               AdditionalAlarms := FALSE,
                               AdditionalWarnings := FALSE);
   END_IF;
   #MachineInterface := "MachineInterface_2_To_1"(MachineInterface_1 := #MachineInterface,
                           MachineInterface_2 := #Sollevatori[4].MachineInterface,
                           AdditionalAlarms := FALSE,
                           AdditionalWarnings := FALSE,
                           ENO => #_w4);
   IF #_w4 THEN
       #MachineInterface := "MachineInterface_2_To_1"(MachineInterface_1 := #MachineInterface,
                               MachineInterface_2 := #Sollevatori[5].MachineInterface,
                               AdditionalAlarms := FALSE,
                               AdditionalWarnings := FALSE);
   END_IF;
   #MachineInterface := "MachineInterface_2_To_1"(MachineInterface_1 := #MachineInterface,
                           MachineInterface_2 := #Sollevatori[6].MachineInterface,
                           AdditionalAlarms := FALSE,
                           AdditionalWarnings := NOT (NOT #Warning.OP_REST_MissingCnd AND NOT #Warning.OP_WORK_MissingCnd));
END_REGION
END_FUNCTION_BLOCK
